LIN {X 0,Y 418.257,Z 234.886,A -85,B 0,C 180,E1 -9993.855,E2 -9993.855} C_VEL
LIN {X 0,Y 418.476,Z 234.858,A -85,B 0,C 180,E1 -9995.784,E2 -9995.784} C_VEL
LIN {X 0,Y 418.364,Z 234.87,A -85,B 0,C 180,E1 -9998.697,E2 -9998.697} C_VEL
LIN {X 0,Y 418.295,Z 234.879,A -85,B 0,C 180,E1 -10001.632,E2 -10001.632} C_VEL
LIN {X 0,Y 418.27,Z 234.881,A -85,B 0,C 180,E1 -10004.599,E2 -10004.599} C_VEL
LIN {X 0,Y 418.253,Z 234.884,A -85,B 0,C 180,E1 -10007.606,E2 -10007.606} C_VEL
LIN {X 0,Y 418.216,Z 234.886,A -85,B 0,C 180,E1 -10010.665,E2 -10010.665} C_VEL
LIN {X 0,Y 418.242,Z 234.885,A -85,B 0,C 180,E1 -10013.785,E2 -10013.785} C_VEL
LIN {X 0,Y 418.196,Z 234.889,A -85,B 0,C 180,E1 -10017.051,E2 -10017.051} C_VEL
LIN {X 0,Y 418.212,Z 234.887,A -85,B 0,C 180,E1 -10020.275,E2 -10020.275} C_VEL
LIN {X 0,Y 418.203,Z 234.887,A -85,B 0,C 180,E1 -10023.682,E2 -10023.682} C_VEL
LIN {X 0,Y 418.207,Z 234.887,A -85,B 0,C 180,E1 -10027.228,E2 -10027.228} C_VEL
LIN {X 0,Y 418.182,Z 234.887,A -85,B 0,C 180,E1 -10030.87,E2 -10030.87} C_VEL
LIN {X 0,Y 418.179,Z 234.883,A -85,B 0,C 180,E1 -10033.732,E2 -10033.732} C_VEL
LIN {X 0,Y 418.178,Z 234.894,A -85,B 0,C 180,E1 -10036.451,E2 -10036.451} C_VEL
LIN {X 0,Y 418.186,Z 234.885,A -85,B 0,C 180,E1 -10039.137,E2 -10039.137} C_VEL
LIN {X 0,Y 418.22,Z 234.877,A -85,B 0,C 180,E1 -10042.779,E2 -10042.779} C_VEL
LIN {X 0,Y 418.216,Z 234.886,A -85,B 0,C 180,E1 -10046.325,E2 -10046.325} C_VEL
LIN {X 0,Y 418.224,Z 234.873,A -85,B 0,C 180,E1 -10049.731,E2 -10049.731} C_VEL
LIN {X 0,Y 418.196,Z 234.877,A -85,B 0,C 180,E1 -10053.02,E2 -10053.02} C_VEL
LIN {X 0,Y 418.245,Z 234.882,A -85,B 0,C 180,E1 -10056.221,E2 -10056.221} C_VEL
LIN {X 0,Y 418.242,Z 234.884,A -85,B 0,C 180,E1 -10059.341,E2 -10059.341} C_VEL
LIN {X 0,Y 418.272,Z 234.856,A -85,B 0,C 180,E1 -10062.4,E2 -10062.4} C_VEL
LIN {X 0,Y 418.295,Z 234.87,A -85,B 0,C 180,E1 -10065.407,E2 -10065.407} C_VEL
LIN {X 0,Y 418.299,Z 234.876,A -85,B 0,C 180,E1 -10068.372,E2 -10068.372} C_VEL
LIN {X 0,Y 418.445,Z 234.844,A -85,B 0,C 180,E1 -10072.282,E2 -10072.282} C_VEL
LIN {X 0,Y 418.469,Z 234.837,A -85,B 0,C 180,E1 -10074.22,E2 -10074.22} C_VEL
LIN {X 0,Y 418.535,Z 234.848,A -85,B 0,C 180,E1 -10078.079,E2 -10078.079} C_VEL
LIN {X 0,Y 418.466,Z 234.853,A -85,B 0,C 180,E1 -10080.966,E2 -10080.966} C_VEL
LIN {X 0,Y 418.471,Z 234.845,A -85,B 0,C 180,E1 -10082.891,E2 -10082.891} C_VEL
LIN {X 0,Y 418.499,Z 234.832,A -85,B 0,C 180,E1 -10085.786,E2 -10085.786} C_VEL
LIN {X 0,Y 418.38,Z 234.87,A -85,B 0,C 180,E1 -10088.699,E2 -10088.699} C_VEL
LIN {X 0,Y 418.317,Z 234.873,A -85,B 0,C 180,E1 -10091.634,E2 -10091.634} C_VEL
LIN {X 0,Y 418.307,Z 234.865,A -85,B 0,C 180,E1 -10094.6,E2 -10094.6} C_VEL
LIN {X 0,Y 418.287,Z 234.874,A -85,B 0,C 180,E1 -10097.607,E2 -10097.607} C_VEL
LIN {X 0,Y 418.258,Z 234.887,A -85,B 0,C 180,E1 -10100.665,E2 -10100.665} C_VEL
LIN {X 0,Y 418.282,Z 234.863,A -85,B 0,C 180,E1 -10103.784,E2 -10103.784} C_VEL
LIN {X 0,Y 418.232,Z 234.889,A -85,B 0,C 180,E1 -10107.048,E2 -10107.048} C_VEL
LIN {X 0,Y 418.252,Z 234.877,A -85,B 0,C 180,E1 -10110.274,E2 -10110.274} C_VEL
LIN {X 0,Y 418.243,Z 234.886,A -85,B 0,C 180,E1 -10113.68,E2 -10113.68} C_VEL
LIN {X 0,Y 418.248,Z 234.881,A -85,B 0,C 180,E1 -10117.226,E2 -10117.226} C_VEL
LIN {X 0,Y 418.219,Z 234.887,A -85,B 0,C 180,E1 -10120.868,E2 -10120.868} C_VEL
LIN {X 0,Y 418.216,Z 234.891,A -85,B 0,C 180,E1 -10123.73,E2 -10123.73} C_VEL
LIN {X 0,Y 418.212,Z 234.885,A -85,B 0,C 180,E1 -10126.448,E2 -10126.448} C_VEL
LIN {X 0,Y 418.219,Z 234.887,A -85,B 0,C 180,E1 -10129.134,E2 -10129.134} C_VEL
LIN {X 0,Y 418.249,Z 234.884,A -85,B 0,C 180,E1 -10132.776,E2 -10132.776} C_VEL
LIN {X 0,Y 418.26,Z 234.88,A -85,B 0,C 180,E1 -10136.323,E2 -10136.323} C_VEL
LIN {X 0,Y 418.256,Z 234.882,A -85,B 0,C 180,E1 -10139.728,E2 -10139.728} C_VEL
LIN {X 0,Y 418.276,Z 234.882,A -85,B 0,C 180,E1 -10143.021,E2 -10143.021} C_VEL
LIN {X 0,Y 418.325,Z 235.179,A -85,B 0,C 180,E1 -10143.563,E2 -10143.563} C_VEL
LIN {X 0,Y 420.735,Z 247.292,A -85,B 0,C 180,E1 -10146.365,E2 -10146.365} C_VEL
LIN {X 0,Y 421.002,Z 250.418,A -85,B 0,C 180,E1 -10147.052,E2 -10147.052} C_VEL
LIN {X 0,Y 419.833,Z 267.822,A -85,B 0,C 180,E1 -10150.693,E2 -10150.693} C_VEL
LIN {X 0,Y 419.789,Z 269.662,A -85,B 0,C 180,E1 -10151.009,E2 -10151.009} C_VEL
LIN {X 0,Y 423.734,Z 293.591,A -85,B 0,C 180,E1 -10151.631,E2 -10151.631} C_VEL
LIN {X 0,Y 422.717,Z 377.028,A -85,B 0,C 180,E1 -10153.084,E2 -10153.084} C_VEL
LIN {X 0,Y 422.229,Z 390.307,A -85,B 0,C 180,E1 -10153.5,E2 -10153.5} C_VEL
LIN {X 0,Y 421.642,Z 403.053,A -85,B 0,C 180,E1 -10154.098,E2 -10154.098} C_VEL
LIN {X 0,Y 420.933,Z 415.178,A -85,B 0,C 180,E1 -10154.877,E2 -10154.877} C_VEL
LIN {X 0,Y 420.162,Z 427.115,A -85,B 0,C 180,E1 -10155.877,E2 -10155.877} C_VEL
LIN {X 0,Y 419.545,Z 437.113,A -85,B 0,C 180,E1 -10156.929,E2 -10156.929} C_VEL
LIN {X 0,Y 418.846,Z 446.446,A -85,B 0,C 180,E1 -10158.138,E2 -10158.138} C_VEL
LIN {X 0,Y 418.173,Z 455.483,A -85,B 0,C 180,E1 -10159.591,E2 -10159.591} C_VEL
LIN {X 0,Y 417.731,Z 462.762,A -85,B 0,C 180,E1 -10161.046,E2 -10161.046} C_VEL
LIN {X 0,Y 417.411,Z 467.677,A -85,B 0,C 180,E1 -10162.258,E2 -10162.258} C_VEL
LIN {X 0,Y 417.167,Z 472.465,A -85,B 0,C 180,E1 -10163.717,E2 -10163.717} C_VEL
LIN {X 0,Y 417.121,Z 476.104,A -85,B 0,C 180,E1 -10165.167,E2 -10165.167} C_VEL
LIN {X 0,Y 417.003,Z 477.99,A -85,B 0,C 180,E1 -10166.134,E2 -10166.134} C_VEL
LIN {X 0,Y 416.987,Z 479.414,A -85,B 0,C 180,E1 -10167.101,E2 -10167.101} C_VEL
LIN {X 0,Y 417.033,Z 480.426,A -85,B 0,C 180,E1 -10168.068,E2 -10168.068} C_VEL
LIN {X 0,Y 416.986,Z 481.283,A -85,B 0,C 180,E1 -10169.999,E2 -10169.999} C_VEL
LIN {X 0,Y 416.996,Z 481.089,A -85,B 0,C 180,E1 -10170.965,E2 -10170.965} C_VEL
LIN {X 0,Y 417.033,Z 480.493,A -85,B 0,C 180,E1 -10171.931,E2 -10171.931} C_VEL
LIN {X 0,Y 417.003,Z 478.128,A -85,B 0,C 180,E1 -10173.865,E2 -10173.865} C_VEL
LIN {X 0,Y 417.162,Z 475.214,A -85,B 0,C 180,E1 -10175.316,E2 -10175.316} C_VEL
LIN {X 0,Y 417.25,Z 471.268,A -85,B 0,C 180,E1 -10176.77,E2 -10176.77} C_VEL
LIN {X 0,Y 417.547,Z 466.19,A -85,B 0,C 180,E1 -10178.225,E2 -10178.225} C_VEL
LIN {X 0,Y 417.934,Z 459.8,A -85,B 0,C 180,E1 -10179.68,E2 -10179.68} C_VEL
LIN {X 0,Y 418.486,Z 451.815,A -85,B 0,C 180,E1 -10181.135,E2 -10181.135} C_VEL
LIN {X 0,Y 419.313,Z 441.896,A -85,B 0,C 180,E1 -10182.584,E2 -10182.584} C_VEL
LIN {X 0,Y 420.026,Z 431.811,A -85,B 0,C 180,E1 -10183.759,E2 -10183.759} C_VEL
LIN {X 0,Y 420.708,Z 421.199,A -85,B 0,C 180,E1 -10184.758,E2 -10184.758} C_VEL
LIN {X 0,Y 421.457,Z 409.943,A -85,B 0,C 180,E1 -10185.597,E2 -10185.597} C_VEL
LIN {X 0,Y 422.163,Z 397.246,A -85,B 0,C 180,E1 -10186.315,E2 -10186.315} C_VEL
LIN {X 0,Y 422.717,Z 383.65,A -85,B 0,C 180,E1 -10186.852,E2 -10186.852} C_VEL
LIN {X 0,Y 423.144,Z 369.847,A -85,B 0,C 180,E1 -10187.176,E2 -10187.176} C_VEL
LIN {X 0,Y 423.875,Z 292.546,A -85,B 0,C 180,E1 -10188.521,E2 -10188.521} C_VEL
LIN {X 0,Y 419.885,Z 269.167,A -85,B 0,C 180,E1 -10189.174,E2 -10189.174} C_VEL
LIN {X 0,Y 420.808,Z 253.629,A -85,B 0,C 180,E1 -10192.33,E2 -10192.33} C_VEL
LIN {X 0,Y 421,Z 248.821,A -85,B 0,C 180,E1 -10193.34,E2 -10193.34} C_VEL
LIN {X 0,Y 418.677,Z 236.536,A -85,B 0,C 180,E1 -10196.143,E2 -10196.143} C_VEL
LIN {X 0,Y 418.322,Z 234.908,A -85,B 0,C 180,E1 -10196.604,E2 -10196.604} C_VEL
LIN {X 0,Y 418.271,Z 234.885,A -85,B 0,C 180,E1 -10199.16,E2 -10199.16} C_VEL
LIN {X 0,Y 418.263,Z 234.884,A -85,B 0,C 180,E1 -10202.842,E2 -10202.842} C_VEL
LIN {X 0,Y 418.248,Z 234.882,A -85,B 0,C 180,E1 -10206.236,E2 -10206.236} C_VEL
LIN {X 0,Y 418.204,Z 234.887,A -85,B 0,C 180,E1 -10209.686,E2 -10209.686} C_VEL
LIN {X 0,Y 418.225,Z 234.891,A -85,B 0,C 180,E1 -10212.318,E2 -10212.318} C_VEL
LIN {X 0,Y 418.237,Z 234.884,A -85,B 0,C 180,E1 -10215.106,E2 -10215.106} C_VEL
LIN {X 0,Y 418.235,Z 234.886,A -85,B 0,C 180,E1 -10217.763,E2 -10217.763} C_VEL
LIN {X 0,Y 418.239,Z 234.88,A -85,B 0,C 180,E1 -10221.554,E2 -10221.554} C_VEL
LIN {X 0,Y 418.251,Z 234.882,A -85,B 0,C 180,E1 -10225.156,E2 -10225.156} C_VEL
LIN {X 0,Y 418.244,Z 234.882,A -85,B 0,C 180,E1 -10227.469,E2 -10227.469} C_VEL
LIN {X 0,Y 418.261,Z 234.885,A -85,B 0,C 180,E1 -10230.895,E2 -10230.895} C_VEL
LIN {X 0,Y 418.217,Z 234.885,A -85,B 0,C 180,E1 -10234.09,E2 -10234.09} C_VEL
LIN {X 0,Y 418.226,Z 234.885,A -85,B 0,C 180,E1 -10237.26,E2 -10237.26} C_VEL
LIN {X 0,Y 418.281,Z 234.879,A -85,B 0,C 180,E1 -10240.361,E2 -10240.361} C_VEL
LIN {X 0,Y 418.313,Z 234.879,A -85,B 0,C 180,E1 -10243.402,E2 -10243.402} C_VEL
LIN {X 0,Y 418.342,Z 234.868,A -85,B 0,C 180,E1 -10246.997,E2 -10246.997} C_VEL
LIN {X 0,Y 418.32,Z 234.872,A -85,B 0,C 180,E1 -10250.325,E2 -10250.325} C_VEL
LIN {X 0,Y 418.459,Z 234.859,A -85,B 0,C 180,E1 -10253.245,E2 -10253.245} C_VEL
LIN {X 0,Y 418.308,Z 234.88,A -85,B 0,C 180,E1 -10255.178,E2 -10255.178} C_VEL
LIN {X 0,Y 418.522,Z 234.85,A -85,B 0,C 180,E1 -10258.072,E2 -10258.072} C_VEL
LIN {X 0,Y 418.52,Z 234.851,A -85,B 0,C 180,E1 -10261.921,E2 -10261.921} C_VEL
LIN {X 0,Y 418.418,Z 234.859,A -85,B 0,C 180,E1 -10266.479,E2 -10266.479} C_VEL
LIN {X 0,Y 418.353,Z 234.868,A -85,B 0,C 180,E1 -10268.692,E2 -10268.692} C_VEL
LIN {X 0,Y 418.338,Z 234.871,A -85,B 0,C 180,E1 -10272.611,E2 -10272.611} C_VEL
LIN {X 0,Y 418.283,Z 234.882,A -85,B 0,C 180,E1 -10275.591,E2 -10275.591} C_VEL
LIN {X 0,Y 418.256,Z 234.885,A -85,B 0,C 180,E1 -10278.614,E2 -10278.614} C_VEL
LIN {X 0,Y 418.215,Z 234.89,A -85,B 0,C 180,E1 -10281.693,E2 -10281.693} C_VEL
LIN {X 0,Y 418.247,Z 234.883,A -85,B 0,C 180,E1 -10284.856,E2 -10284.856} C_VEL
LIN {X 0,Y 418.226,Z 234.886,A -85,B 0,C 180,E1 -10288.063,E2 -10288.063} C_VEL
LIN {X 0,Y 418.187,Z 234.89,A -85,B 0,C 180,E1 -10291.393,E2 -10291.393} C_VEL
LIN {X 0,Y 418.241,Z 234.886,A -85,B 0,C 180,E1 -10294.577,E2 -10294.577} C_VEL
LIN {X 0,Y 418.211,Z 234.888,A -85,B 0,C 180,E1 -10297.832,E2 -10297.832} C_VEL
LIN {X 0,Y 418.239,Z 234.888,A -85,B 0,C 180,E1 -10300.94,E2 -10300.94} C_VEL
LIN {X 0,Y 418.303,Z 235.044,A -85,B 0,C 180,E1 -10302.724,E2 -10302.724} C_VEL
LIN {X 0,Y 420.273,Z 244.859,A -85,B 0,C 180,E1 -10305.027,E2 -10305.027} C_VEL
LIN {X 0,Y 420.476,Z 249.038,A -85,B 0,C 180,E1 -10305.942,E2 -10305.942} C_VEL
LIN {X 0,Y 419.996,Z 258.446,A -85,B 0,C 180,E1 -10307.877,E2 -10307.877} C_VEL
LIN {X 0,Y 424.024,Z 279.663,A -85,B 0,C 180,E1 -10308.495,E2 -10308.495} C_VEL
LIN {X 0,Y 422.987,Z 365.547,A -85,B 0,C 180,E1 -10310.001,E2 -10310.001} C_VEL
LIN {X 0,Y 422.557,Z 379.31,A -85,B 0,C 180,E1 -10310.436,E2 -10310.436} C_VEL
LIN {X 0,Y 422.008,Z 392.261,A -85,B 0,C 180,E1 -10311.053,E2 -10311.053} C_VEL
LIN {X 0,Y 421.307,Z 404.921,A -85,B 0,C 180,E1 -10311.888,E2 -10311.888} C_VEL
LIN {X 0,Y 420.52,Z 416.351,A -85,B 0,C 180,E1 -10312.863,E2 -10312.863} C_VEL
LIN {X 0,Y 419.798,Z 425.954,A -85,B 0,C 180,E1 -10313.883,E2 -10313.883} C_VEL
LIN {X 0,Y 419.22,Z 434.271,A -85,B 0,C 180,E1 -10314.959,E2 -10314.959} C_VEL
LIN {X 0,Y 418.541,Z 443.069,A -85,B 0,C 180,E1 -10316.351,E2 -10316.351} C_VEL
LIN {X 0,Y 417.991,Z 450.165,A -85,B 0,C 180,E1 -10317.736,E2 -10317.736} C_VEL
LIN {X 0,Y 417.595,Z 456.913,A -85,B 0,C 180,E1 -10319.392,E2 -10319.392} C_VEL
LIN {X 0,Y 417.253,Z 462.266,A -85,B 0,C 180,E1 -10321.137,E2 -10321.137} C_VEL
LIN {X 0,Y 416.99,Z 466.192,A -85,B 0,C 180,E1 -10322.932,E2 -10322.932} C_VEL
LIN {X 0,Y 416.899,Z 467.831,A -85,B 0,C 180,E1 -10324.006,E2 -10324.006} C_VEL
LIN {X 0,Y 416.837,Z 469.291,A -85,B 0,C 180,E1 -10325.556,E2 -10325.556} C_VEL
LIN {X 0,Y 416.773,Z 469.714,A -85,B 0,C 180,E1 -10327.18,E2 -10327.18} C_VEL
LIN {X 0,Y 416.83,Z 469.386,A -85,B 0,C 180,E1 -10328.228,E2 -10328.228} C_VEL
LIN {X 0,Y 416.837,Z 468.631,A -85,B 0,C 180,E1 -10329.265,E2 -10329.265} C_VEL
LIN {X 0,Y 416.982,Z 466.785,A -85,B 0,C 180,E1 -10330.693,E2 -10330.693} C_VEL
LIN {X 0,Y 417.16,Z 463.519,A -85,B 0,C 180,E1 -10332.348,E2 -10332.348} C_VEL
LIN {X 0,Y 417.403,Z 458.75,A -85,B 0,C 180,E1 -10334.039,E2 -10334.039} C_VEL
LIN {X 0,Y 417.787,Z 452.809,A -85,B 0,C 180,E1 -10335.634,E2 -10335.634} C_VEL
LIN {X 0,Y 418.218,Z 446.156,A -85,B 0,C 180,E1 -10337.053,E2 -10337.053} C_VEL
LIN {X 0,Y 418.742,Z 438.489,A -85,B 0,C 180,E1 -10338.382,E2 -10338.382} C_VEL
LIN {X 0,Y 419.451,Z 428.69,A -85,B 0,C 180,E1 -10339.746,E2 -10339.746} C_VEL
LIN {X 0,Y 420.123,Z 419.264,A -85,B 0,C 180,E1 -10340.811,E2 -10340.811} C_VEL
LIN {X 0,Y 419.772,Z 414.556,A -85,B 0,C 180,E1 -10341.294,E2 -10341.294} C_VEL
LIN {X 0,Y 417.471,Z 406.719,A -85,B 0,C 180,E1 -10342.063,E2 -10342.063} C_VEL
LIN {X 0,Y 415.262,Z 398.464,A -85,B 0,C 180,E1 -10342.761,E2 -10342.761} C_VEL
LIN {X 0,Y 414.864,Z 393.162,A -85,B 0,C 180,E1 -10343.118,E2 -10343.118} C_VEL
LIN {X 0,Y 415.338,Z 382.041,A -85,B 0,C 180,E1 -10343.686,E2 -10343.686} C_VEL
LIN {X 0,Y 415.835,Z 368.781,A -85,B 0,C 180,E1 -10344.15,E2 -10344.15} C_VEL
LIN {X 0,Y 416.183,Z 350.094,A -85,B 0,C 180,E1 -10344.522,E2 -10344.522} C_VEL
LIN {X 0,Y 416.884,Z 280.038,A -85,B 0,C 180,E1 -10345.753,E2 -10345.753} C_VEL
LIN {X 0,Y 412.979,Z 258.958,A -85,B 0,C 180,E1 -10346.342,E2 -10346.342} C_VEL
LIN {X 0,Y 413.209,Z 254.351,A -85,B 0,C 180,E1 -10347.32,E2 -10347.32} C_VEL
LIN {X 0,Y 413.524,Z 247.973,A -85,B 0,C 180,E1 -10348.784,E2 -10348.784} C_VEL
LIN {X 0,Y 412.086,Z 239.005,A -85,B 0,C 180,E1 -10350.978,E2 -10350.978} C_VEL
LIN {X 0,Y 411.483,Z 235.781,A -85,B 0,C 180,E1 -10351.836,E2 -10351.836} C_VEL
LIN {X 0,Y 411.438,Z 235.734,A -85,B 0,C 180,E1 -10355.883,E2 -10355.883} C_VEL
LIN {X 0,Y 411.319,Z 235.748,A -85,B 0,C 180,E1 -10358.847,E2 -10358.847} C_VEL
LIN {X 0,Y 411.263,Z 235.752,A -85,B 0,C 180,E1 -10361.834,E2 -10361.834} C_VEL
LIN {X 0,Y 411.226,Z 235.758,A -85,B 0,C 180,E1 -10364.855,E2 -10364.855} C_VEL
LIN {X 0,Y 411.218,Z 235.765,A -85,B 0,C 180,E1 -10367.917,E2 -10367.917} C_VEL
LIN {X 0,Y 411.163,Z 235.764,A -85,B 0,C 180,E1 -10371.037,E2 -10371.037} C_VEL
LIN {X 0,Y 411.18,Z 235.763,A -85,B 0,C 180,E1 -10374.219,E2 -10374.219} C_VEL
LIN {X 0,Y 411.158,Z 235.767,A -85,B 0,C 180,E1 -10377.486,E2 -10377.486} C_VEL
LIN {X 0,Y 411.159,Z 235.766,A -85,B 0,C 180,E1 -10380.851,E2 -10380.851} C_VEL
LIN {X 0,Y 411.164,Z 235.762,A -85,B 0,C 180,E1 -10384.338,E2 -10384.338} C_VEL
LIN {X 0,Y 411.159,Z 235.768,A -85,B 0,C 180,E1 -10386.746,E2 -10386.746} C_VEL
LIN {X 0,Y 411.142,Z 235.768,A -85,B 0,C 180,E1 -10389.723,E2 -10389.723} C_VEL
LIN {X 0,Y 411.139,Z 235.762,A -85,B 0,C 180,E1 -10393.139,E2 -10393.139} C_VEL
LIN {X 0,Y 411.142,Z 235.767,A -85,B 0,C 180,E1 -10395.885,E2 -10395.885} C_VEL
LIN {X 0,Y 411.138,Z 235.76,A -85,B 0,C 180,E1 -10399.497,E2 -10399.497} C_VEL
LIN {X 0,Y 411.168,Z 235.75,A -85,B 0,C 180,E1 -10402.029,E2 -10402.029} C_VEL
LIN {X 0,Y 411.186,Z 235.767,A -85,B 0,C 180,E1 -10405.127,E2 -10405.127} C_VEL
LIN {X 0,Y 411.148,Z 235.763,A -85,B 0,C 180,E1 -10408.006,E2 -10408.006} C_VEL
LIN {X 0,Y 411.158,Z 235.75,A -85,B 0,C 180,E1 -10411.41,E2 -10411.41} C_VEL
LIN {X 0,Y 411.177,Z 235.761,A -85,B 0,C 180,E1 -10414.945,E2 -10414.945} C_VEL
LIN {X 0,Y 411.194,Z 235.761,A -85,B 0,C 180,E1 -10417.917,E2 -10417.917} C_VEL
LIN {X 0,Y 411.211,Z 235.749,A -85,B 0,C 180,E1 -10421.055,E2 -10421.055} C_VEL
LIN {X 0,Y 411.247,Z 235.746,A -85,B 0,C 180,E1 -10424.135,E2 -10424.135} C_VEL
LIN {X 0,Y 411.298,Z 235.747,A -85,B 0,C 180,E1 -10427.169,E2 -10427.169} C_VEL
LIN {X 0,Y 411.276,Z 235.749,A -85,B 0,C 180,E1 -10430.165,E2 -10430.165} C_VEL
LIN {X 0,Y 411.389,Z 235.719,A -85,B 0,C 180,E1 -10433.135,E2 -10433.135} C_VEL
LIN {X 0,Y 411.287,Z 235.731,A -85,B 0,C 180,E1 -10435.102,E2 -10435.102} C_VEL
LIN {X 0,Y 411.504,Z 235.723,A -85,B 0,C 180,E1 -10438.046,E2 -10438.046} C_VEL
LIN {X 0,Y 411.431,Z 235.729,A -85,B 0,C 180,E1 -10440.982,E2 -10440.982} C_VEL
LIN {X 0,Y 411.429,Z 235.722,A -85,B 0,C 180,E1 -10442.941,E2 -10442.941} C_VEL
LIN {X 0,Y 411.435,Z 235.726,A -85,B 0,C 180,E1 -10446.87,E2 -10446.87} C_VEL
LIN {X 0,Y 411.289,Z 235.749,A -85,B 0,C 180,E1 -10449.842,E2 -10449.842} C_VEL
LIN {X 0,Y 411.313,Z 235.74,A -85,B 0,C 180,E1 -10453.106,E2 -10453.106} C_VEL
LIN {X 0,Y 411.266,Z 235.747,A -85,B 0,C 180,E1 -10456.891,E2 -10456.891} C_VEL
LIN {X 0,Y 411.24,Z 235.756,A -85,B 0,C 180,E1 -10459.989,E2 -10459.989} C_VEL
LIN {X 0,Y 411.204,Z 235.75,A -85,B 0,C 180,E1 -10463.15,E2 -10463.15} C_VEL
LIN {X 0,Y 411.195,Z 235.758,A -85,B 0,C 180,E1 -10466.387,E2 -10466.387} C_VEL
LIN {X 0,Y 411.207,Z 235.756,A -85,B 0,C 180,E1 -10469.715,E2 -10469.715} C_VEL
LIN {X 0,Y 411.215,Z 235.759,A -85,B 0,C 180,E1 -10473.158,E2 -10473.158} C_VEL
LIN {X 0,Y 411.202,Z 235.757,A -85,B 0,C 180,E1 -10476.554,E2 -10476.554} C_VEL
LIN {X 0,Y 411.18,Z 235.768,A -85,B 0,C 180,E1 -10479.722,E2 -10479.722} C_VEL
LIN {X 0,Y 411.176,Z 235.759,A -85,B 0,C 180,E1 -10483.136,E2 -10483.136} C_VEL
LIN {X 0,Y 411.175,Z 235.765,A -85,B 0,C 180,E1 -10485.883,E2 -10485.883} C_VEL
LIN {X 0,Y 411.16,Z 235.765,A -85,B 0,C 180,E1 -10488.775,E2 -10488.775} C_VEL
LIN {X 0,Y 411.197,Z 235.765,A -85,B 0,C 180,E1 -10492.026,E2 -10492.026} C_VEL
LIN {X 0,Y 411.217,Z 235.763,A -85,B 0,C 180,E1 -10495.667,E2 -10495.667} C_VEL
LIN {X 0,Y 411.201,Z 235.761,A -85,B 0,C 180,E1 -10499.153,E2 -10499.153} C_VEL
LIN {X 0,Y 411.254,Z 235.761,A -85,B 0,C 180,E1 -10502.521,E2 -10502.521} C_VEL
LIN {X 0,Y 411.304,Z 235.978,A -85,B 0,C 180,E1 -10503.286,E2 -10503.286} C_VEL
LIN {X 0,Y 413.93,Z 249.498,A -85,B 0,C 180,E1 -10506.473,E2 -10506.473} C_VEL
LIN {X 0,Y 413.717,Z 255.587,A -85,B 0,C 180,E1 -10507.791,E2 -10507.791} C_VEL
LIN {X 0,Y 412.851,Z 269.407,A -85,B 0,C 180,E1 -10510.677,E2 -10510.677} C_VEL
LIN {X 0,Y 414.868,Z 281.394,A -85,B 0,C 180,E1 -10511.022,E2 -10511.022} C_VEL
LIN {X 0,Y 416.982,Z 294.541,A -85,B 0,C 180,E1 -10511.355,E2 -10511.355} C_VEL
LIN {X 0,Y 415.893,Z 377.561,A -85,B 0,C 180,E1 -10512.83,E2 -10512.83} C_VEL
LIN {X 0,Y 415.331,Z 391.388,A -85,B 0,C 180,E1 -10513.281,E2 -10513.281} C_VEL
LIN {X 0,Y 414.745,Z 403.809,A -85,B 0,C 180,E1 -10513.889,E2 -10513.889} C_VEL
LIN {X 0,Y 413.955,Z 416.487,A -85,B 0,C 180,E1 -10514.742,E2 -10514.742} C_VEL
LIN {X 0,Y 413.223,Z 427.367,A -85,B 0,C 180,E1 -10515.683,E2 -10515.683} C_VEL
LIN {X 0,Y 412.534,Z 437.926,A -85,B 0,C 180,E1 -10516.828,E2 -10516.828} C_VEL
LIN {X 0,Y 411.715,Z 447.892,A -85,B 0,C 180,E1 -10518.179,E2 -10518.179} C_VEL
LIN {X 0,Y 411.084,Z 456.668,A -85,B 0,C 180,E1 -10519.658,E2 -10519.658} C_VEL
LIN {X 0,Y 410.607,Z 463.663,A -85,B 0,C 180,E1 -10521.138,E2 -10521.138} C_VEL
LIN {X 0,Y 410.285,Z 469.262,A -85,B 0,C 180,E1 -10522.618,E2 -10522.618} C_VEL
LIN {X 0,Y 410.063,Z 473.658,A -85,B 0,C 180,E1 -10524.097,E2 -10524.097} C_VEL
LIN {X 0,Y 410.035,Z 475.98,A -85,B 0,C 180,E1 -10525.083,E2 -10525.083} C_VEL
LIN {X 0,Y 409.923,Z 477.872,A -85,B 0,C 180,E1 -10526.067,E2 -10526.067} C_VEL
LIN {X 0,Y 409.886,Z 479.303,A -85,B 0,C 180,E1 -10527.051,E2 -10527.051} C_VEL
LIN {X 0,Y 409.93,Z 480.319,A -85,B 0,C 180,E1 -10528.034,E2 -10528.034} C_VEL
LIN {X 0,Y 409.922,Z 480.945,A -85,B 0,C 180,E1 -10529.017,E2 -10529.017} C_VEL
LIN {X 0,Y 409.91,Z 481.183,A -85,B 0,C 180,E1 -10529.999,E2 -10529.999} C_VEL
LIN {X 0,Y 409.922,Z 480.996,A -85,B 0,C 180,E1 -10530.982,E2 -10530.982} C_VEL
LIN {X 0,Y 409.929,Z 480.403,A -85,B 0,C 180,E1 -10531.964,E2 -10531.964} C_VEL
LIN {X 0,Y 409.925,Z 478.046,A -85,B 0,C 180,E1 -10533.931,E2 -10533.931} C_VEL
LIN {X 0,Y 410.079,Z 475.138,A -85,B 0,C 180,E1 -10535.408,E2 -10535.408} C_VEL
LIN {X 0,Y 410.187,Z 471.199,A -85,B 0,C 180,E1 -10536.888,E2 -10536.888} C_VEL
LIN {X 0,Y 410.493,Z 466.128,A -85,B 0,C 180,E1 -10538.367,E2 -10538.367} C_VEL
LIN {X 0,Y 410.905,Z 459.751,A -85,B 0,C 180,E1 -10539.847,E2 -10539.847} C_VEL
LIN {X 0,Y 411.514,Z 451.775,A -85,B 0,C 180,E1 -10541.326,E2 -10541.326} C_VEL
LIN {X 0,Y 412.383,Z 441.868,A -85,B 0,C 180,E1 -10542.799,E2 -10542.799} C_VEL
LIN {X 0,Y 413.097,Z 431.339,A -85,B 0,C 180,E1 -10544.045,E2 -10544.045} C_VEL
LIN {X 0,Y 413.862,Z 421.211,A -85,B 0,C 180,E1 -10545.008,E2 -10545.008} C_VEL
LIN {X 0,Y 414.614,Z 409.981,A -85,B 0,C 180,E1 -10545.862,E2 -10545.862} C_VEL
LIN {X 0,Y 415.367,Z 397.349,A -85,B 0,C 180,E1 -10546.589,E2 -10546.589} C_VEL
LIN {X 0,Y 415.955,Z 383.839,A -85,B 0,C 180,E1 -10547.134,E2 -10547.134} C_VEL
LIN {X 0,Y 416.384,Z 370.314,A -85,B 0,C 180,E1 -10547.464,E2 -10547.464} C_VEL
LIN {X 0,Y 417.199,Z 293.585,A -85,B 0,C 180,E1 -10548.82,E2 -10548.82} C_VEL
LIN {X 0,Y 412.997,Z 269.348,A -85,B 0,C 180,E1 -10549.498,E2 -10549.498} C_VEL
LIN {X 0,Y 413.044,Z 267.047,A -85,B 0,C 180,E1 -10549.894,E2 -10549.894} C_VEL
LIN {X 0,Y 414.064,Z 252.374,A -85,B 0,C 180,E1 -10552.977,E2 -10552.977} C_VEL
LIN {X 0,Y 413.881,Z 248.977,A -85,B 0,C 180,E1 -10553.724,E2 -10553.724} C_VEL
LIN {X 0,Y 411.307,Z 235.976,A -85,B 0,C 180,E1 -10556.783,E2 -10556.783} C_VEL
LIN {X 0,Y 411.206,Z 235.763,A -85,B 0,C 180,E1 -10559.711,E2 -10559.711} C_VEL
LIN {X 0,Y 411.212,Z 235.763,A -85,B 0,C 180,E1 -10563.154,E2 -10563.154} C_VEL
LIN {X 0,Y 411.196,Z 235.759,A -85,B 0,C 180,E1 -10566.55,E2 -10566.55} C_VEL
LIN {X 0,Y 411.173,Z 235.763,A -85,B 0,C 180,E1 -10569.718,E2 -10569.718} C_VEL
LIN {X 0,Y 411.173,Z 235.763,A -85,B 0,C 180,E1 -10573.132,E2 -10573.132} C_VEL
LIN {X 0,Y 411.17,Z 235.766,A -85,B 0,C 180,E1 -10575.879,E2 -10575.879} C_VEL
LIN {X 0,Y 411.155,Z 235.77,A -85,B 0,C 180,E1 -10578.771,E2 -10578.771} C_VEL
LIN {X 0,Y 411.187,Z 235.761,A -85,B 0,C 180,E1 -10582.023,E2 -10582.023} C_VEL
LIN {X 0,Y 411.204,Z 235.76,A -85,B 0,C 180,E1 -10585.121,E2 -10585.121} C_VEL
LIN {X 0,Y 411.165,Z 235.765,A -85,B 0,C 180,E1 -10588,E2 -10588} C_VEL
LIN {X 0,Y 411.175,Z 235.763,A -85,B 0,C 180,E1 -10591.404,E2 -10591.404} C_VEL
LIN {X 0,Y 411.187,Z 235.768,A -85,B 0,C 180,E1 -10594.938,E2 -10594.938} C_VEL
LIN {X 0,Y 411.201,Z 235.757,A -85,B 0,C 180,E1 -10597.91,E2 -10597.91} C_VEL
LIN {X 0,Y 411.216,Z 235.758,A -85,B 0,C 180,E1 -10601.048,E2 -10601.048} C_VEL
LIN {X 0,Y 411.248,Z 235.755,A -85,B 0,C 180,E1 -10604.129,E2 -10604.129} C_VEL
LIN {X 0,Y 411.299,Z 235.747,A -85,B 0,C 180,E1 -10607.163,E2 -10607.163} C_VEL
LIN {X 0,Y 411.275,Z 235.749,A -85,B 0,C 180,E1 -10610.158,E2 -10610.158} C_VEL
LIN {X 0,Y 411.425,Z 235.734,A -85,B 0,C 180,E1 -10613.129,E2 -10613.129} C_VEL
LIN {X 0,Y 411.281,Z 235.754,A -85,B 0,C 180,E1 -10615.095,E2 -10615.095} C_VEL
LIN {X 0,Y 411.491,Z 235.726,A -85,B 0,C 180,E1 -10618.039,E2 -10618.039} C_VEL
LIN {X 0,Y 411.489,Z 235.727,A -85,B 0,C 180,E1 -10621.954,E2 -10621.954} C_VEL
LIN {X 0,Y 411.368,Z 235.737,A -85,B 0,C 180,E1 -10626.477,E2 -10626.477} C_VEL
LIN {X 0,Y 411.293,Z 235.748,A -85,B 0,C 180,E1 -10628.843,E2 -10628.843} C_VEL
LIN {X 0,Y 411.259,Z 235.76,A -85,B 0,C 180,E1 -10631.83,E2 -10631.83} C_VEL
LIN {X 0,Y 411.241,Z 235.757,A -85,B 0,C 180,E1 -10634.849,E2 -10634.849} C_VEL
LIN {X 0,Y 411.227,Z 235.76,A -85,B 0,C 180,E1 -10637.912,E2 -10637.912} C_VEL
LIN {X 0,Y 411.177,Z 235.764,A -85,B 0,C 180,E1 -10641.031,E2 -10641.031} C_VEL
LIN {X 0,Y 411.192,Z 235.768,A -85,B 0,C 180,E1 -10644.213,E2 -10644.213} C_VEL
LIN {X 0,Y 411.167,Z 235.766,A -85,B 0,C 180,E1 -10647.48,E2 -10647.48} C_VEL
LIN {X 0,Y 411.165,Z 235.768,A -85,B 0,C 180,E1 -10650.845,E2 -10650.845} C_VEL
LIN {X 0,Y 411.181,Z 235.767,A -85,B 0,C 180,E1 -10654.33,E2 -10654.33} C_VEL
LIN {X 0,Y 411.178,Z 235.765,A -85,B 0,C 180,E1 -10657.97,E2 -10657.97} C_VEL
LIN {X 0,Y 411.183,Z 235.768,A -85,B 0,C 180,E1 -10661.233,E2 -10661.233} C_VEL
LIN {X 0,Y 411.256,Z 235.96,A -85,B 0,C 180,E1 -10662.452,E2 -10662.452} C_VEL
LIN {X 0,Y 413.507,Z 247.488,A -85,B 0,C 180,E1 -10665.194,E2 -10665.194} C_VEL
LIN {X 0,Y 413.299,Z 254.821,A -85,B 0,C 180,E1 -10666.781,E2 -10666.781} C_VEL
LIN {X 0,Y 413.17,Z 258.636,A -85,B 0,C 180,E1 -10667.537,E2 -10667.537} C_VEL
LIN {X 0,Y 417.351,Z 280.584,A -85,B 0,C 180,E1 -10668.19,E2 -10668.19} C_VEL
LIN {X 0,Y 416.189,Z 366.364,A -85,B 0,C 180,E1 -10669.723,E2 -10669.723} C_VEL
LIN {X 0,Y 415.757,Z 380.018,A -85,B 0,C 180,E1 -10670.172,E2 -10670.172} C_VEL
LIN {X 0,Y 415.23,Z 392.101,A -85,B 0,C 180,E1 -10670.76,E2 -10670.76} C_VEL
LIN {X 0,Y 414.629,Z 403.053,A -85,B 0,C 180,E1 -10671.472,E2 -10671.472} C_VEL
LIN {X 0,Y 413.787,Z 414.416,A -85,B 0,C 180,E1 -10672.419,E2 -10672.419} C_VEL
LIN {X 0,Y 412.93,Z 425.552,A -85,B 0,C 180,E1 -10673.591,E2 -10673.591} C_VEL
LIN {X 0,Y 412.184,Z 435.562,A -85,B 0,C 180,E1 -10674.919,E2 -10674.919} C_VEL
LIN {X 0,Y 411.487,Z 443.872,A -85,B 0,C 180,E1 -10676.285,E2 -10676.285} C_VEL
LIN {X 0,Y 410.931,Z 450.847,A -85,B 0,C 180,E1 -10677.694,E2 -10677.694} C_VEL
LIN {X 0,Y 410.565,Z 456.474,A -85,B 0,C 180,E1 -10679.102,E2 -10679.102} C_VEL
LIN {X 0,Y 410.206,Z 462.03,A -85,B 0,C 180,E1 -10680.89,E2 -10680.89} C_VEL
LIN {X 0,Y 410.012,Z 465.535,A -85,B 0,C 180,E1 -10682.433,E2 -10682.433} C_VEL
LIN {X 0,Y 409.837,Z 467.351,A -85,B 0,C 180,E1 -10683.523,E2 -10683.523} C_VEL
LIN {X 0,Y 409.734,Z 469.303,A -85,B 0,C 180,E1 -10685.367,E2 -10685.367} C_VEL
LIN {X 0,Y 409.693,Z 469.807,A -85,B 0,C 180,E1 -10686.763,E2 -10686.763} C_VEL
LIN {X 0,Y 409.692,Z 469.672,A -85,B 0,C 180,E1 -10687.857,E2 -10687.857} C_VEL
LIN {X 0,Y 409.73,Z 469.06,A -85,B 0,C 180,E1 -10688.888,E2 -10688.888} C_VEL
LIN {X 0,Y 409.869,Z 467.155,A -85,B 0,C 180,E1 -10690.56,E2 -10690.56} C_VEL
LIN {X 0,Y 410.019,Z 464.481,A -85,B 0,C 180,E1 -10692.03,E2 -10692.03} C_VEL
LIN {X 0,Y 410.218,Z 460.513,A -85,B 0,C 180,E1 -10693.601,E2 -10693.601} C_VEL
LIN {X 0,Y 410.555,Z 455.461,A -85,B 0,C 180,E1 -10695.122,E2 -10695.122} C_VEL
LIN {X 0,Y 410.997,Z 449.104,A -85,B 0,C 180,E1 -10696.635,E2 -10696.635} C_VEL
LIN {X 0,Y 411.584,Z 440.919,A -85,B 0,C 180,E1 -10698.177,E2 -10698.177} C_VEL
LIN {X 0,Y 412.207,Z 432.636,A -85,B 0,C 180,E1 -10699.44,E2 -10699.44} C_VEL
LIN {X 0,Y 413.001,Z 422.379,A -85,B 0,C 180,E1 -10700.712,E2 -10700.712} C_VEL
LIN {X 0,Y 413.796,Z 411.053,A -85,B 0,C 180,E1 -10701.823,E2 -10701.823} C_VEL
LIN {X 0,Y 414.549,Z 399.759,A -85,B 0,C 180,E1 -10702.696,E2 -10702.696} C_VEL
LIN {X 0,Y 414.864,Z 393.162,A -85,B 0,C 180,E1 -10703.118,E2 -10703.118} C_VEL
LIN {X 0,Y 414.381,Z 389.563,A -85,B 0,C 180,E1 -10703.354,E2 -10703.354} C_VEL
LIN {X 0,Y 409.267,Z 378.214,A -85,B 0,C 180,E1 -10704.099,E2 -10704.099} C_VEL
LIN {X 0,Y 408.871,Z 374.429,A -85,B 0,C 180,E1 -10704.255,E2 -10704.255} C_VEL
LIN {X 0,Y 409.232,Z 361.718,A -85,B 0,C 180,E1 -10704.599,E2 -10704.599} C_VEL
LIN {X 0,Y 410.187,Z 281.4,A -85,B 0,C 180,E1 -10706.032,E2 -10706.032} C_VEL
LIN {X 0,Y 406.081,Z 259.104,A -85,B 0,C 180,E1 -10706.662,E2 -10706.662} C_VEL
LIN {X 0,Y 406.283,Z 255.054,A -85,B 0,C 180,E1 -10707.522,E2 -10707.522} C_VEL
LIN {X 0,Y 406.518,Z 248.699,A -85,B 0,C 180,E1 -10709.01,E2 -10709.01} C_VEL
LIN {X 0,Y 405.213,Z 240.733,A -85,B 0,C 180,E1 -10710.995,E2 -10710.995} C_VEL
LIN {X 0,Y 404.449,Z 236.659,A -85,B 0,C 180,E1 -10712.086,E2 -10712.086} C_VEL
LIN {X 0,Y 404.386,Z 236.612,A -85,B 0,C 180,E1 -10715.986,E2 -10715.986} C_VEL
LIN {X 0,Y 404.256,Z 236.627,A -85,B 0,C 180,E1 -10719.003,E2 -10719.003} C_VEL
LIN {X 0,Y 404.234,Z 236.625,A -85,B 0,C 180,E1 -10722.043,E2 -10722.043} C_VEL
LIN {X 0,Y 404.172,Z 236.638,A -85,B 0,C 180,E1 -10725.12,E2 -10725.12} C_VEL
LIN {X 0,Y 404.176,Z 236.638,A -85,B 0,C 180,E1 -10728.24,E2 -10728.24} C_VEL
LIN {X 0,Y 404.105,Z 236.645,A -85,B 0,C 180,E1 -10731.422,E2 -10731.422} C_VEL
LIN {X 0,Y 404.132,Z 236.64,A -85,B 0,C 180,E1 -10734.669,E2 -10734.669} C_VEL
LIN {X 0,Y 404.1,Z 236.647,A -85,B 0,C 180,E1 -10738.008,E2 -10738.008} C_VEL
LIN {X 0,Y 404.115,Z 236.642,A -85,B 0,C 180,E1 -10740.288,E2 -10740.288} C_VEL
LIN {X 0,Y 404.11,Z 236.644,A -85,B 0,C 180,E1 -10743.816,E2 -10743.816} C_VEL
LIN {X 0,Y 404.105,Z 236.646,A -85,B 0,C 180,E1 -10746.877,E2 -10746.877} C_VEL
LIN {X 0,Y 404.092,Z 236.648,A -85,B 0,C 180,E1 -10750.078,E2 -10750.078} C_VEL
LIN {X 0,Y 404.118,Z 236.636,A -85,B 0,C 180,E1 -10753.086,E2 -10753.086} C_VEL
LIN {X 0,Y 404.098,Z 236.644,A -85,B 0,C 180,E1 -10755.926,E2 -10755.926} C_VEL
LIN {X 0,Y 404.082,Z 236.65,A -85,B 0,C 180,E1 -10758.636,E2 -10758.636} C_VEL
LIN {X 0,Y 404.122,Z 236.629,A -85,B 0,C 180,E1 -10761.499,E2 -10761.499} C_VEL
LIN {X 0,Y 404.158,Z 236.64,A -85,B 0,C 180,E1 -10764.987,E2 -10764.987} C_VEL
LIN {X 0,Y 404.122,Z 236.638,A -85,B 0,C 180,E1 -10768.447,E2 -10768.447} C_VEL
LIN {X 0,Y 404.135,Z 236.625,A -85,B 0,C 180,E1 -10770.866,E2 -10770.866} C_VEL
LIN {X 0,Y 404.143,Z 236.635,A -85,B 0,C 180,E1 -10774.727,E2 -10774.727} C_VEL
LIN {X 0,Y 404.157,Z 236.642,A -85,B 0,C 180,E1 -10777.512,E2 -10777.512} C_VEL
LIN {X 0,Y 404.155,Z 236.626,A -85,B 0,C 180,E1 -10780.711,E2 -10780.711} C_VEL
LIN {X 0,Y 404.215,Z 236.616,A -85,B 0,C 180,E1 -10783.852,E2 -10783.852} C_VEL
LIN {X 0,Y 404.28,Z 236.62,A -85,B 0,C 180,E1 -10786.943,E2 -10786.943} C_VEL
LIN {X 0,Y 404.243,Z 236.627,A -85,B 0,C 180,E1 -10789.992,E2 -10789.992} C_VEL
LIN {X 0,Y 404.34,Z 236.597,A -85,B 0,C 180,E1 -10793.015,E2 -10793.015} C_VEL
LIN {X 0,Y 404.258,Z 236.606,A -85,B 0,C 180,E1 -10795.017,E2 -10795.017} C_VEL
LIN {X 0,Y 404.473,Z 236.598,A -85,B 0,C 180,E1 -10798.012,E2 -10798.012} C_VEL
LIN {X 0,Y 404.397,Z 236.605,A -85,B 0,C 180,E1 -10800.999,E2 -10800.999} C_VEL
LIN {X 0,Y 404.363,Z 236.602,A -85,B 0,C 180,E1 -10802.992,E2 -10802.992} C_VEL
LIN {X 0,Y 404.396,Z 236.589,A -85,B 0,C 180,E1 -10805.989,E2 -10805.989} C_VEL
LIN {X 0,Y 404.267,Z 236.625,A -85,B 0,C 180,E1 -10809.005,E2 -10809.005} C_VEL
LIN {X 0,Y 404.261,Z 236.625,A -85,B 0,C 180,E1 -10812.044,E2 -10812.044} C_VEL
LIN {X 0,Y 404.211,Z 236.616,A -85,B 0,C 180,E1 -10815.121,E2 -10815.121} C_VEL
LIN {X 0,Y 404.213,Z 236.628,A -85,B 0,C 180,E1 -10818.241,E2 -10818.241} C_VEL
LIN {X 0,Y 404.147,Z 236.637,A -85,B 0,C 180,E1 -10821.422,E2 -10821.422} C_VEL
LIN {X 0,Y 404.17,Z 236.624,A -85,B 0,C 180,E1 -10824.669,E2 -10824.669} C_VEL
LIN {X 0,Y 404.13,Z 236.641,A -85,B 0,C 180,E1 -10828.007,E2 -10828.007} C_VEL
LIN {X 0,Y 404.154,Z 236.633,A -85,B 0,C 180,E1 -10830.287,E2 -10830.287} C_VEL
LIN {X 0,Y 404.149,Z 236.641,A -85,B 0,C 180,E1 -10833.815,E2 -10833.815} C_VEL
LIN {X 0,Y 404.145,Z 236.638,A -85,B 0,C 180,E1 -10836.876,E2 -10836.876} C_VEL
LIN {X 0,Y 404.128,Z 236.643,A -85,B 0,C 180,E1 -10840.076,E2 -10840.076} C_VEL
LIN {X 0,Y 404.156,Z 236.633,A -85,B 0,C 180,E1 -10843.083,E2 -10843.083} C_VEL
LIN {X 0,Y 404.132,Z 236.642,A -85,B 0,C 180,E1 -10845.923,E2 -10845.923} C_VEL
LIN {X 0,Y 404.115,Z 236.643,A -85,B 0,C 180,E1 -10848.634,E2 -10848.634} C_VEL
LIN {X 0,Y 404.151,Z 236.643,A -85,B 0,C 180,E1 -10851.496,E2 -10851.496} C_VEL
LIN {X 0,Y 404.196,Z 236.635,A -85,B 0,C 180,E1 -10854.984,E2 -10854.984} C_VEL
LIN {X 0,Y 404.151,Z 236.642,A -85,B 0,C 180,E1 -10858.443,E2 -10858.443} C_VEL
LIN {X 0,Y 404.199,Z 236.635,A -85,B 0,C 180,E1 -10862,E2 -10862} C_VEL
LIN {X 0,Y 404.251,Z 236.853,A -85,B 0,C 180,E1 -10863.023,E2 -10863.023} C_VEL
LIN {X 0,Y 406.647,Z 248.969,A -85,B 0,C 180,E1 -10865.948,E2 -10865.948} C_VEL
LIN {X 0,Y 407.081,Z 252.998,A -85,B 0,C 180,E1 -10866.873,E2 -10866.873} C_VEL
LIN {X 0,Y 405.938,Z 269.125,A -85,B 0,C 180,E1 -10870.335,E2 -10870.335} C_VEL
LIN {X 0,Y 406.589,Z 273.393,A -85,B 0,C 180,E1 -10870.496,E2 -10870.496} C_VEL
LIN {X 0,Y 410.2,Z 295.407,A -85,B 0,C 180,E1 -10871.068,E2 -10871.068} C_VEL
LIN {X 0,Y 409.118,Z 376.957,A -85,B 0,C 180,E1 -10872.537,E2 -10872.537} C_VEL
LIN {X 0,Y 408.598,Z 390.189,A -85,B 0,C 180,E1 -10872.965,E2 -10872.965} C_VEL
LIN {X 0,Y 407.917,Z 403.47,A -85,B 0,C 180,E1 -10873.612,E2 -10873.612} C_VEL
LIN {X 0,Y 407.18,Z 414.624,A -85,B 0,C 180,E1 -10874.353,E2 -10874.353} C_VEL
LIN {X 0,Y 406.364,Z 426.617,A -85,B 0,C 180,E1 -10875.386,E2 -10875.386} C_VEL
LIN {X 0,Y 405.631,Z 436.675,A -85,B 0,C 180,E1 -10876.472,E2 -10876.472} C_VEL
LIN {X 0,Y 404.898,Z 446.069,A -85,B 0,C 180,E1 -10877.723,E2 -10877.723} C_VEL
LIN {X 0,Y 404.146,Z 455.138,A -85,B 0,C 180,E1 -10879.225,E2 -10879.225} C_VEL
LIN {X 0,Y 403.626,Z 462.444,A -85,B 0,C 180,E1 -10880.731,E2 -10880.731} C_VEL
LIN {X 0,Y 403.307,Z 467.386,A -85,B 0,C 180,E1 -10881.986,E2 -10881.986} C_VEL
LIN {X 0,Y 402.988,Z 472.961,A -85,B 0,C 180,E1 -10883.767,E2 -10883.767} C_VEL
LIN {X 0,Y 402.95,Z 475.855,A -85,B 0,C 180,E1 -10884.996,E2 -10884.996} C_VEL
LIN {X 0,Y 402.846,Z 477.751,A -85,B 0,C 180,E1 -10885.998,E2 -10885.998} C_VEL
LIN {X 0,Y 402.788,Z 479.191,A -85,B 0,C 180,E1 -10886.999,E2 -10886.999} C_VEL
LIN {X 0,Y 402.826,Z 480.211,A -85,B 0,C 180,E1 -10888,E2 -10888} C_VEL
LIN {X 0,Y 402.849,Z 480.841,A -85,B 0,C 180,E1 -10889,E2 -10889} C_VEL
LIN {X 0,Y 402.836,Z 481.084,A -85,B 0,C 180,E1 -10889.999,E2 -10889.999} C_VEL
LIN {X 0,Y 402.849,Z 480.903,A -85,B 0,C 180,E1 -10890.999,E2 -10890.999} C_VEL
LIN {X 0,Y 402.826,Z 480.313,A -85,B 0,C 180,E1 -10891.999,E2 -10891.999} C_VEL
LIN {X 0,Y 402.849,Z 477.963,A -85,B 0,C 180,E1 -10894.001,E2 -10894.001} C_VEL
LIN {X 0,Y 402.976,Z 475.062,A -85,B 0,C 180,E1 -10895.503,E2 -10895.503} C_VEL
LIN {X 0,Y 403.11,Z 471.129,A -85,B 0,C 180,E1 -10897.009,E2 -10897.009} C_VEL
LIN {X 0,Y 403.453,Z 466.066,A -85,B 0,C 180,E1 -10898.514,E2 -10898.514} C_VEL
LIN {X 0,Y 403.888,Z 459.7,A -85,B 0,C 180,E1 -10900.02,E2 -10900.02} C_VEL
LIN {X 0,Y 404.536,Z 451.735,A -85,B 0,C 180,E1 -10901.524,E2 -10901.524} C_VEL
LIN {X 0,Y 405.44,Z 441.84,A -85,B 0,C 180,E1 -10903.022,E2 -10903.022} C_VEL
LIN {X 0,Y 406.137,Z 432.299,A -85,B 0,C 180,E1 -10904.186,E2 -10904.186} C_VEL
LIN {X 0,Y 406.877,Z 422.665,A -85,B 0,C 180,E1 -10905.144,E2 -10905.144} C_VEL
LIN {X 0,Y 407.702,Z 411.816,A -85,B 0,C 180,E1 -10906.009,E2 -10906.009} C_VEL
LIN {X 0,Y 408.409,Z 399.861,A -85,B 0,C 180,E1 -10906.751,E2 -10906.751} C_VEL
LIN {X 0,Y 409.098,Z 386.854,A -85,B 0,C 180,E1 -10907.334,E2 -10907.334} C_VEL
LIN {X 0,Y 409.529,Z 373.962,A -85,B 0,C 180,E1 -10907.701,E2 -10907.701} C_VEL
LIN {X 0,Y 410.541,Z 294.671,A -85,B 0,C 180,E1 -10909.131,E2 -10909.131} C_VEL
LIN {X 0,Y 406.32,Z 270.523,A -85,B 0,C 180,E1 -10909.807,E2 -10909.807} C_VEL
LIN {X 0,Y 406.063,Z 268.841,A -85,B 0,C 180,E1 -10909.897,E2 -10909.897} C_VEL
LIN {X 0,Y 407.163,Z 253.578,A -85,B 0,C 180,E1 -10913.121,E2 -10913.121} C_VEL
LIN {X 0,Y 406.772,Z 249.447,A -85,B 0,C 180,E1 -10914.056,E2 -10914.056} C_VEL
LIN {X 0,Y 404.436,Z 237.713,A -85,B 0,C 180,E1 -10916.859,E2 -10916.859} C_VEL
LIN {X 0,Y 404.251,Z 236.662,A -85,B 0,C 180,E1 -10917.186,E2 -10917.186} C_VEL
LIN {X 0,Y 404.151,Z 236.644,A -85,B 0,C 180,E1 -10920.283,E2 -10920.283} C_VEL
LIN {X 0,Y 404.15,Z 236.64,A -85,B 0,C 180,E1 -10923.81,E2 -10923.81} C_VEL
LIN {X 0,Y 404.139,Z 236.638,A -85,B 0,C 180,E1 -10926.872,E2 -10926.872} C_VEL
LIN {X 0,Y 404.121,Z 236.639,A -85,B 0,C 180,E1 -10930.073,E2 -10930.073} C_VEL
LIN {X 0,Y 404.153,Z 236.637,A -85,B 0,C 180,E1 -10933.081,E2 -10933.081} C_VEL
LIN {X 0,Y 404.15,Z 236.641,A -85,B 0,C 180,E1 -10935.923,E2 -10935.923} C_VEL
LIN {X 0,Y 404.11,Z 236.646,A -85,B 0,C 180,E1 -10938.631,E2 -10938.631} C_VEL
LIN {X 0,Y 404.142,Z 236.636,A -85,B 0,C 180,E1 -10941.492,E2 -10941.492} C_VEL
LIN {X 0,Y 404.175,Z 236.636,A -85,B 0,C 180,E1 -10944.98,E2 -10944.98} C_VEL
LIN {X 0,Y 404.139,Z 236.641,A -85,B 0,C 180,E1 -10948.44,E2 -10948.44} C_VEL
LIN {X 0,Y 404.151,Z 236.643,A -85,B 0,C 180,E1 -10950.86,E2 -10950.86} C_VEL
LIN {X 0,Y 404.152,Z 236.643,A -85,B 0,C 180,E1 -10954.72,E2 -10954.72} C_VEL
LIN {X 0,Y 404.165,Z 236.635,A -85,B 0,C 180,E1 -10957.505,E2 -10957.505} C_VEL
LIN {X 0,Y 404.159,Z 236.641,A -85,B 0,C 180,E1 -10960.704,E2 -10960.704} C_VEL
LIN {X 0,Y 404.216,Z 236.631,A -85,B 0,C 180,E1 -10963.845,E2 -10963.845} C_VEL
LIN {X 0,Y 404.279,Z 236.619,A -85,B 0,C 180,E1 -10966.936,E2 -10966.936} C_VEL
LIN {X 0,Y 404.242,Z 236.626,A -85,B 0,C 180,E1 -10969.985,E2 -10969.985} C_VEL
LIN {X 0,Y 404.375,Z 236.61,A -85,B 0,C 180,E1 -10973.009,E2 -10973.009} C_VEL
LIN {X 0,Y 404.254,Z 236.629,A -85,B 0,C 180,E1 -10975.01,E2 -10975.01} C_VEL
LIN {X 0,Y 404.46,Z 236.602,A -85,B 0,C 180,E1 -10978.005,E2 -10978.005} C_VEL
LIN {X 0,Y 404.458,Z 236.603,A -85,B 0,C 180,E1 -10981.988,E2 -10981.988} C_VEL
LIN {X 0,Y 404.321,Z 236.615,A -85,B 0,C 180,E1 -10986.474,E2 -10986.474} C_VEL
LIN {X 0,Y 404.242,Z 236.626,A -85,B 0,C 180,E1 -10988.998,E2 -10988.998} C_VEL
LIN {X 0,Y 404.234,Z 236.633,A -85,B 0,C 180,E1 -10992.038,E2 -10992.038} C_VEL
LIN {X 0,Y 404.188,Z 236.636,A -85,B 0,C 180,E1 -10995.115,E2 -10995.115} C_VEL
LIN {X 0,Y 404.186,Z 236.641,A -85,B 0,C 180,E1 -10998.235,E2 -10998.235} C_VEL
LIN {X 0,Y 404.119,Z 236.644,A -85,B 0,C 180,E1 -11001.416,E2 -11001.416} C_VEL
LIN {X 0,Y 404.144,Z 236.641,A -85,B 0,C 180,E1 -11004.663,E2 -11004.663} C_VEL
LIN {X 0,Y 404.108,Z 236.644,A -85,B 0,C 180,E1 -11008.001,E2 -11008.001} C_VEL
LIN {X 0,Y 404.121,Z 236.647,A -85,B 0,C 180,E1 -11010.282,E2 -11010.282} C_VEL
LIN {X 0,Y 404.121,Z 236.646,A -85,B 0,C 180,E1 -11013.809,E2 -11013.809} C_VEL
LIN {X 0,Y 404.114,Z 236.646,A -85,B 0,C 180,E1 -11016.873,E2 -11016.873} C_VEL
LIN {X 0,Y 404.14,Z 236.645,A -85,B 0,C 180,E1 -11020.081,E2 -11020.081} C_VEL
LIN {X 0,Y 404.206,Z 236.72,A -85,B 0,C 180,E1 -11022.099,E2 -11022.099} C_VEL
LIN {X 0,Y 405.278,Z 242.084,A -85,B 0,C 180,E1 -11023.462,E2 -11023.462} C_VEL
LIN {X 0,Y 406.688,Z 250.081,A -85,B 0,C 180,E1 -11025.346,E2 -11025.346} C_VEL
LIN {X 0,Y 406.272,Z 258.551,A -85,B 0,C 180,E1 -11027.151,E2 -11027.151} C_VEL
LIN {X 0,Y 407.057,Z 262.671,A -85,B 0,C 180,E1 -11027.327,E2 -11027.327} C_VEL
LIN {X 0,Y 410.711,Z 282.156,A -85,B 0,C 180,E1 -11027.885,E2 -11027.885} C_VEL
LIN {X 0,Y 409.457,Z 366.408,A -85,B 0,C 180,E1 -11029.412,E2 -11029.412} C_VEL
LIN {X 0,Y 409,Z 379.932,A -85,B 0,C 180,E1 -11029.862,E2 -11029.862} C_VEL
LIN {X 0,Y 408.466,Z 392.062,A -85,B 0,C 180,E1 -11030.462,E2 -11030.462} C_VEL
LIN {X 0,Y 407.795,Z 403.521,A -85,B 0,C 180,E1 -11031.221,E2 -11031.221} C_VEL
LIN {X 0,Y 406.901,Z 414.826,A -85,B 0,C 180,E1 -11032.184,E2 -11032.184} C_VEL
LIN {X 0,Y 406.041,Z 425.557,A -85,B 0,C 180,E1 -11033.336,E2 -11033.336} C_VEL
LIN {X 0,Y 405.307,Z 434.872,A -85,B 0,C 180,E1 -11034.577,E2 -11034.577} C_VEL
LIN {X 0,Y 404.589,Z 443.134,A -85,B 0,C 180,E1 -11035.931,E2 -11035.931} C_VEL
LIN {X 0,Y 403.965,Z 450.255,A -85,B 0,C 180,E1 -11037.364,E2 -11037.364} C_VEL
LIN {X 0,Y 403.495,Z 457.115,A -85,B 0,C 180,E1 -11039.102,E2 -11039.102} C_VEL
LIN {X 0,Y 403.138,Z 462.161,A -85,B 0,C 180,E1 -11040.783,E2 -11040.783} C_VEL
LIN {X 0,Y 402.962,Z 464.77,A -85,B 0,C 180,E1 -11041.908,E2 -11041.908} C_VEL
LIN {X 0,Y 402.808,Z 466.834,A -85,B 0,C 180,E1 -11043.024,E2 -11043.024} C_VEL
LIN {X 0,Y 402.699,Z 468.317,A -85,B 0,C 180,E1 -11044.133,E2 -11044.133} C_VEL
LIN {X 0,Y 402.636,Z 469.331,A -85,B 0,C 180,E1 -11045.235,E2 -11045.235} C_VEL
LIN {X 0,Y 402.597,Z 469.841,A -85,B 0,C 180,E1 -11046.329,E2 -11046.329} C_VEL
LIN {X 0,Y 402.596,Z 469.824,A -85,B 0,C 180,E1 -11047.686,E2 -11047.686} C_VEL
LIN {X 0,Y 402.674,Z 468.565,A -85,B 0,C 180,E1 -11049.571,E2 -11049.571} C_VEL
LIN {X 0,Y 402.786,Z 467.208,A -85,B 0,C 180,E1 -11050.64,E2 -11050.64} C_VEL
LIN {X 0,Y 402.951,Z 464.314,A -85,B 0,C 180,E1 -11052.229,E2 -11052.229} C_VEL
LIN {X 0,Y 403.186,Z 460.316,A -85,B 0,C 180,E1 -11053.807,E2 -11053.807} C_VEL
LIN {X 0,Y 403.544,Z 455.113,A -85,B 0,C 180,E1 -11055.374,E2 -11055.374} C_VEL
LIN {X 0,Y 404.034,Z 448.536,A -85,B 0,C 180,E1 -11056.932,E2 -11056.932} C_VEL
LIN {X 0,Y 404.641,Z 440.295,A -85,B 0,C 180,E1 -11058.479,E2 -11058.479} C_VEL
LIN {X 0,Y 405.295,Z 431.875,A -85,B 0,C 180,E1 -11059.763,E2 -11059.763} C_VEL
LIN {X 0,Y 406.122,Z 421.534,A -85,B 0,C 180,E1 -11061.041,E2 -11061.041} C_VEL
LIN {X 0,Y 406.898,Z 411.224,A -85,B 0,C 180,E1 -11062.059,E2 -11062.059} C_VEL
LIN {X 0,Y 407.676,Z 399.948,A -85,B 0,C 180,E1 -11062.945,E2 -11062.945} C_VEL
LIN {X 0,Y 408.285,Z 387.509,A -85,B 0,C 180,E1 -11063.701,E2 -11063.701} C_VEL
LIN {X 0,Y 408.871,Z 374.429,A -85,B 0,C 180,E1 -11064.255,E2 -11064.255} C_VEL
LIN {X 0,Y 408.662,Z 368.708,A -85,B 0,C 180,E1 -11064.452,E2 -11064.452} C_VEL
LIN {X 0,Y 406.097,Z 359.421,A -85,B 0,C 180,E1 -11064.78,E2 -11064.78} C_VEL
LIN {X 0,Y 403.333,Z 350.079,A -85,B 0,C 180,E1 -11065.075,E2 -11065.075} C_VEL
LIN {X 0,Y 402.699,Z 344.257,A -85,B 0,C 180,E1 -11065.208,E2 -11065.208} C_VEL
LIN {X 0,Y 403.457,Z 282.291,A -85,B 0,C 180,E1 -11066.332,E2 -11066.332} C_VEL
LIN {X 0,Y 399.159,Z 259.085,A -85,B 0,C 180,E1 -11067.005,E2 -11067.005} C_VEL
LIN {X 0,Y 399.624,Z 250.439,A -85,B 0,C 180,E1 -11068.993,E2 -11068.993} C_VEL
LIN {X 0,Y 398.333,Z 242.457,A -85,B 0,C 180,E1 -11071.012,E2 -11071.012} C_VEL
LIN {X 0,Y 397.394,Z 237.542,A -85,B 0,C 180,E1 -11072.345,E2 -11072.345} C_VEL
LIN {X 0,Y 397.337,Z 237.489,A -85,B 0,C 180,E1 -11076.093,E2 -11076.093} C_VEL
LIN {X 0,Y 397.218,Z 237.503,A -85,B 0,C 180,E1 -11079.163,E2 -11079.163} C_VEL
LIN {X 0,Y 397.194,Z 237.5,A -85,B 0,C 180,E1 -11082.26,E2 -11082.26} C_VEL
LIN {X 0,Y 397.145,Z 237.515,A -85,B 0,C 180,E1 -11085.394,E2 -11085.394} C_VEL
LIN {X 0,Y 397.128,Z 237.514,A -85,B 0,C 180,E1 -11088.576,E2 -11088.576} C_VEL
LIN {X 0,Y 397.063,Z 237.526,A -85,B 0,C 180,E1 -11091.821,E2 -11091.821} C_VEL
LIN {X 0,Y 397.092,Z 237.516,A -85,B 0,C 180,E1 -11095.137,E2 -11095.137} C_VEL
LIN {X 0,Y 397.048,Z 237.518,A -85,B 0,C 180,E1 -11098.55,E2 -11098.55} C_VEL
LIN {X 0,Y 397.052,Z 237.525,A -85,B 0,C 180,E1 -11101.839,E2 -11101.839} C_VEL
LIN {X 0,Y 397.089,Z 237.512,A -85,B 0,C 180,E1 -11104.498,E2 -11104.498} C_VEL
LIN {X 0,Y 397.064,Z 237.525,A -85,B 0,C 180,E1 -11108.28,E2 -11108.28} C_VEL
LIN {X 0,Y 397.027,Z 237.518,A -85,B 0,C 180,E1 -11111.98,E2 -11111.98} C_VEL
LIN {X 0,Y 397.063,Z 237.524,A -85,B 0,C 180,E1 -11115.073,E2 -11115.073} C_VEL
LIN {X 0,Y 397.031,Z 237.525,A -85,B 0,C 180,E1 -11118.028,E2 -11118.028} C_VEL
LIN {X 0,Y 397.074,Z 237.505,A -85,B 0,C 180,E1 -11121.728,E2 -11121.728} C_VEL
LIN {X 0,Y 397.101,Z 237.519,A -85,B 0,C 180,E1 -11125.51,E2 -11125.51} C_VEL
LIN {X 0,Y 397.062,Z 237.515,A -85,B 0,C 180,E1 -11129.121,E2 -11129.121} C_VEL
LIN {X 0,Y 397.048,Z 237.506,A -85,B 0,C 180,E1 -11132.256,E2 -11132.256} C_VEL
LIN {X 0,Y 397.092,Z 237.514,A -85,B 0,C 180,E1 -11134.869,E2 -11134.869} C_VEL
LIN {X 0,Y 397.086,Z 237.516,A -85,B 0,C 180,E1 -11138.185,E2 -11138.185} C_VEL
LIN {X 0,Y 397.15,Z 237.493,A -85,B 0,C 180,E1 -11141.43,E2 -11141.43} C_VEL
LIN {X 0,Y 397.173,Z 237.497,A -85,B 0,C 180,E1 -11144.612,E2 -11144.612} C_VEL
LIN {X 0,Y 397.211,Z 237.508,A -85,B 0,C 180,E1 -11147.746,E2 -11147.746} C_VEL
LIN {X 0,Y 397.227,Z 237.495,A -85,B 0,C 180,E1 -11150.841,E2 -11150.841} C_VEL
LIN {X 0,Y 397.32,Z 237.469,A -85,B 0,C 180,E1 -11153.911,E2 -11153.911} C_VEL
LIN {X 0,Y 397.441,Z 237.473,A -85,B 0,C 180,E1 -11157.977,E2 -11157.977} C_VEL
LIN {X 0,Y 397.44,Z 237.475,A -85,B 0,C 180,E1 -11162.03,E2 -11162.03} C_VEL
LIN {X 0,Y 397.349,Z 237.467,A -85,B 0,C 180,E1 -11166.095,E2 -11166.095} C_VEL
LIN {X 0,Y 397.238,Z 237.5,A -85,B 0,C 180,E1 -11169.165,E2 -11169.165} C_VEL
LIN {X 0,Y 397.225,Z 237.504,A -85,B 0,C 180,E1 -11172.261,E2 -11172.261} C_VEL
LIN {X 0,Y 397.185,Z 237.49,A -85,B 0,C 180,E1 -11175.395,E2 -11175.395} C_VEL
LIN {X 0,Y 397.166,Z 237.509,A -85,B 0,C 180,E1 -11178.576,E2 -11178.576} C_VEL
LIN {X 0,Y 397.105,Z 237.513,A -85,B 0,C 180,E1 -11181.821,E2 -11181.821} C_VEL
LIN {X 0,Y 397.117,Z 237.508,A -85,B 0,C 180,E1 -11185.137,E2 -11185.137} C_VEL
LIN {X 0,Y 397.082,Z 237.521,A -85,B 0,C 180,E1 -11188.55,E2 -11188.55} C_VEL
LIN {X 0,Y 397.091,Z 237.513,A -85,B 0,C 180,E1 -11191.838,E2 -11191.838} C_VEL
LIN {X 0,Y 397.13,Z 237.514,A -85,B 0,C 180,E1 -11194.496,E2 -11194.496} C_VEL
LIN {X 0,Y 397.103,Z 237.513,A -85,B 0,C 180,E1 -11198.278,E2 -11198.278} C_VEL
LIN {X 0,Y 397.065,Z 237.517,A -85,B 0,C 180,E1 -11201.978,E2 -11201.978} C_VEL
LIN {X 0,Y 397.096,Z 237.52,A -85,B 0,C 180,E1 -11205.07,E2 -11205.07} C_VEL
LIN {X 0,Y 397.065,Z 237.525,A -85,B 0,C 180,E1 -11208.024,E2 -11208.024} C_VEL
LIN {X 0,Y 397.103,Z 237.521,A -85,B 0,C 180,E1 -11211.724,E2 -11211.724} C_VEL
LIN {X 0,Y 397.137,Z 237.517,A -85,B 0,C 180,E1 -11215.507,E2 -11215.507} C_VEL
LIN {X 0,Y 397.09,Z 237.518,A -85,B 0,C 180,E1 -11219.118,E2 -11219.118} C_VEL
LIN {X 0,Y 397.176,Z 237.586,A -85,B 0,C 180,E1 -11222.679,E2 -11222.679} C_VEL
LIN {X 0,Y 398.67,Z 245.016,A -85,B 0,C 180,E1 -11224.568,E2 -11224.568} C_VEL
LIN {X 0,Y 400.106,Z 252.825,A -85,B 0,C 180,E1 -11226.445,E2 -11226.445} C_VEL
LIN {X 0,Y 399.202,Z 266.094,A -85,B 0,C 180,E1 -11229.383,E2 -11229.383} C_VEL
LIN {X 0,Y 399.027,Z 269.39,A -85,B 0,C 180,E1 -11230.034,E2 -11230.034} C_VEL
LIN {X 0,Y 403.372,Z 295.357,A -85,B 0,C 180,E1 -11230.753,E2 -11230.753} C_VEL
LIN {X 0,Y 402.318,Z 377.424,A -85,B 0,C 180,E1 -11232.264,E2 -11232.264} C_VEL
LIN {X 0,Y 401.711,Z 391.23,A -85,B 0,C 180,E1 -11232.73,E2 -11232.73} C_VEL
LIN {X 0,Y 401.04,Z 404.151,A -85,B 0,C 180,E1 -11233.389,E2 -11233.389} C_VEL
LIN {X 0,Y 400.23,Z 415.922,A -85,B 0,C 180,E1 -11234.205,E2 -11234.205} C_VEL
LIN {X 0,Y 399.361,Z 427.795,A -85,B 0,C 180,E1 -11235.268,E2 -11235.268} C_VEL
LIN {X 0,Y 398.539,Z 438.502,A -85,B 0,C 180,E1 -11236.488,E2 -11236.488} C_VEL
LIN {X 0,Y 397.774,Z 447.515,A -85,B 0,C 180,E1 -11237.759,E2 -11237.759} C_VEL
LIN {X 0,Y 397.038,Z 456.326,A -85,B 0,C 180,E1 -11239.288,E2 -11239.288} C_VEL
LIN {X 0,Y 396.536,Z 463.358,A -85,B 0,C 180,E1 -11240.821,E2 -11240.821} C_VEL
LIN {X 0,Y 396.162,Z 468.98,A -85,B 0,C 180,E1 -11242.353,E2 -11242.353} C_VEL
LIN {X 0,Y 395.867,Z 474.047,A -85,B 0,C 180,E1 -11244.151,E2 -11244.151} C_VEL
LIN {X 0,Y 395.771,Z 477.63,A -85,B 0,C 180,E1 -11245.926,E2 -11245.926} C_VEL
LIN {X 0,Y 395.695,Z 479.079,A -85,B 0,C 180,E1 -11246.945,E2 -11246.945} C_VEL
LIN {X 0,Y 395.723,Z 480.102,A -85,B 0,C 180,E1 -11247.964,E2 -11247.964} C_VEL
LIN {X 0,Y 395.761,Z 480.737,A -85,B 0,C 180,E1 -11248.982,E2 -11248.982} C_VEL
LIN {X 0,Y 395.764,Z 480.984,A -85,B 0,C 180,E1 -11249.999,E2 -11249.999} C_VEL
LIN {X 0,Y 395.76,Z 480.81,A -85,B 0,C 180,E1 -11251.017,E2 -11251.017} C_VEL
LIN {X 0,Y 395.723,Z 480.224,A -85,B 0,C 180,E1 -11252.035,E2 -11252.035} C_VEL
LIN {X 0,Y 395.775,Z 477.881,A -85,B 0,C 180,E1 -11254.072,E2 -11254.072} C_VEL
LIN {X 0,Y 395.876,Z 474.986,A -85,B 0,C 180,E1 -11255.602,E2 -11255.602} C_VEL
LIN {X 0,Y 396.061,Z 471.061,A -85,B 0,C 180,E1 -11257.134,E2 -11257.134} C_VEL
LIN {X 0,Y 396.401,Z 466.007,A -85,B 0,C 180,E1 -11258.667,E2 -11258.667} C_VEL
LIN {X 0,Y 396.886,Z 459.659,A -85,B 0,C 180,E1 -11260.199,E2 -11260.199} C_VEL
LIN {X 0,Y 397.541,Z 451.713,A -85,B 0,C 180,E1 -11261.729,E2 -11261.729} C_VEL
LIN {X 0,Y 398.514,Z 441.84,A -85,B 0,C 180,E1 -11263.253,E2 -11263.253} C_VEL
LIN {X 0,Y 399.308,Z 431.533,A -85,B 0,C 180,E1 -11264.522,E2 -11264.522} C_VEL
LIN {X 0,Y 400.164,Z 421.302,A -85,B 0,C 180,E1 -11265.534,E2 -11265.534} C_VEL
LIN {X 0,Y 400.988,Z 410.152,A -85,B 0,C 180,E1 -11266.416,E2 -11266.416} C_VEL
LIN {X 0,Y 401.785,Z 397.709,A -85,B 0,C 180,E1 -11267.167,E2 -11267.167} C_VEL
LIN {X 0,Y 402.451,Z 384.444,A -85,B 0,C 180,E1 -11267.728,E2 -11267.728} C_VEL
LIN {X 0,Y 402.891,Z 371.58,A -85,B 0,C 180,E1 -11268.069,E2 -11268.069} C_VEL
LIN {X 0,Y 403.895,Z 295.759,A -85,B 0,C 180,E1 -11269.453,E2 -11269.453} C_VEL
LIN {X 0,Y 399.808,Z 272.247,A -85,B 0,C 180,E1 -11270.123,E2 -11270.123} C_VEL
LIN {X 0,Y 399.186,Z 268.945,A -85,B 0,C 180,E1 -11270.252,E2 -11270.252} C_VEL
LIN {X 0,Y 400.26,Z 254.796,A -85,B 0,C 180,E1 -11273.269,E2 -11273.269} C_VEL
LIN {X 0,Y 399.662,Z 249.901,A -85,B 0,C 180,E1 -11274.407,E2 -11274.407} C_VEL
LIN {X 0,Y 397.473,Z 238.91,A -85,B 0,C 180,E1 -11277.083,E2 -11277.083} C_VEL
LIN {X 0,Y 397.204,Z 237.531,A -85,B 0,C 180,E1 -11277.531,E2 -11277.531} C_VEL
LIN {X 0,Y 397.084,Z 237.523,A -85,B 0,C 180,E1 -11280.881,E2 -11280.881} C_VEL
LIN {X 0,Y 397.13,Z 237.517,A -85,B 0,C 180,E1 -11284.491,E2 -11284.491} C_VEL
LIN {X 0,Y 397.096,Z 237.523,A -85,B 0,C 180,E1 -11288.274,E2 -11288.274} C_VEL
LIN {X 0,Y 397.062,Z 237.526,A -85,B 0,C 180,E1 -11291.975,E2 -11291.975} C_VEL
LIN {X 0,Y 397.089,Z 237.519,A -85,B 0,C 180,E1 -11295.067,E2 -11295.067} C_VEL
LIN {X 0,Y 397.061,Z 237.526,A -85,B 0,C 180,E1 -11298.02,E2 -11298.02} C_VEL
LIN {X 0,Y 397.094,Z 237.515,A -85,B 0,C 180,E1 -11301.721,E2 -11301.721} C_VEL
LIN {X 0,Y 397.118,Z 237.513,A -85,B 0,C 180,E1 -11305.503,E2 -11305.503} C_VEL
LIN {X 0,Y 397.078,Z 237.521,A -85,B 0,C 180,E1 -11309.115,E2 -11309.115} C_VEL
LIN {X 0,Y 397.063,Z 237.522,A -85,B 0,C 180,E1 -11312.249,E2 -11312.249} C_VEL
LIN {X 0,Y 397.102,Z 237.523,A -85,B 0,C 180,E1 -11314.862,E2 -11314.862} C_VEL
LIN {X 0,Y 397.093,Z 237.515,A -85,B 0,C 180,E1 -11318.178,E2 -11318.178} C_VEL
LIN {X 0,Y 397.155,Z 237.505,A -85,B 0,C 180,E1 -11321.423,E2 -11321.423} C_VEL
LIN {X 0,Y 397.173,Z 237.51,A -85,B 0,C 180,E1 -11324.605,E2 -11324.605} C_VEL
LIN {X 0,Y 397.213,Z 237.504,A -85,B 0,C 180,E1 -11327.739,E2 -11327.739} C_VEL
LIN {X 0,Y 397.223,Z 237.502,A -85,B 0,C 180,E1 -11330.834,E2 -11330.834} C_VEL
LIN {X 0,Y 397.34,Z 237.489,A -85,B 0,C 180,E1 -11333.905,E2 -11333.905} C_VEL
LIN {X 0,Y 397.427,Z 237.479,A -85,B 0,C 180,E1 -11337.97,E2 -11337.97} C_VEL
LIN {X 0,Y 397.425,Z 237.479,A -85,B 0,C 180,E1 -11342.023,E2 -11342.023} C_VEL
LIN {X 0,Y 397.278,Z 237.493,A -85,B 0,C 180,E1 -11346.468,E2 -11346.468} C_VEL
LIN {X 0,Y 397.213,Z 237.503,A -85,B 0,C 180,E1 -11349.159,E2 -11349.159} C_VEL
LIN {X 0,Y 397.199,Z 237.507,A -85,B 0,C 180,E1 -11352.255,E2 -11352.255} C_VEL
LIN {X 0,Y 397.161,Z 237.512,A -85,B 0,C 180,E1 -11355.389,E2 -11355.389} C_VEL
LIN {X 0,Y 397.139,Z 237.516,A -85,B 0,C 180,E1 -11358.57,E2 -11358.57} C_VEL
LIN {X 0,Y 397.077,Z 237.524,A -85,B 0,C 180,E1 -11361.815,E2 -11361.815} C_VEL
LIN {X 0,Y 397.102,Z 237.516,A -85,B 0,C 180,E1 -11365.131,E2 -11365.131} C_VEL
LIN {X 0,Y 397.056,Z 237.519,A -85,B 0,C 180,E1 -11368.544,E2 -11368.544} C_VEL
LIN {X 0,Y 397.058,Z 237.522,A -85,B 0,C 180,E1 -11371.833,E2 -11371.833} C_VEL
LIN {X 0,Y 397.101,Z 237.519,A -85,B 0,C 180,E1 -11374.49,E2 -11374.49} C_VEL
LIN {X 0,Y 397.083,Z 237.523,A -85,B 0,C 180,E1 -11378.271,E2 -11378.271} C_VEL
LIN {X 0,Y 397.147,Z 237.665,A -85,B 0,C 180,E1 -11381.826,E2 -11381.826} C_VEL
LIN {X 0,Y 399.513,Z 249.293,A -85,B 0,C 180,E1 -11384.714,E2 -11384.714} C_VEL
LIN {X 0,Y 399.702,Z 253.993,A -85,B 0,C 180,E1 -11385.791,E2 -11385.791} C_VEL
LIN {X 0,Y 399.448,Z 258.886,A -85,B 0,C 180,E1 -11386.803,E2 -11386.803} C_VEL
LIN {X 0,Y 402.128,Z 272.24,A -85,B 0,C 180,E1 -11387.246,E2 -11387.246} C_VEL
LIN {X 0,Y 404.046,Z 282.636,A -85,B 0,C 180,E1 -11387.547,E2 -11387.547} C_VEL
LIN {X 0,Y 402.759,Z 366.326,A -85,B 0,C 180,E1 -11389.089,E2 -11389.089} C_VEL
LIN {X 0,Y 402.257,Z 379.861,A -85,B 0,C 180,E1 -11389.543,E2 -11389.543} C_VEL
LIN {X 0,Y 401.666,Z 392.676,A -85,B 0,C 180,E1 -11390.188,E2 -11390.188} C_VEL
LIN {X 0,Y 400.891,Z 404.886,A -85,B 0,C 180,E1 -11391.031,E2 -11391.031} C_VEL
LIN {X 0,Y 399.961,Z 416.344,A -85,B 0,C 180,E1 -11392.049,E2 -11392.049} C_VEL
LIN {X 0,Y 399.045,Z 426.792,A -85,B 0,C 180,E1 -11393.217,E2 -11393.217} C_VEL
LIN {X 0,Y 398.344,Z 435.317,A -85,B 0,C 180,E1 -11394.395,E2 -11394.395} C_VEL
LIN {X 0,Y 397.525,Z 444.376,A -85,B 0,C 180,E1 -11395.935,E2 -11395.935} C_VEL
LIN {X 0,Y 396.838,Z 452.21,A -85,B 0,C 180,E1 -11397.608,E2 -11397.608} C_VEL
LIN {X 0,Y 396.416,Z 457.6,A -85,B 0,C 180,E1 -11399.061,E2 -11399.061} C_VEL
LIN {X 0,Y 396.04,Z 462.77,A -85,B 0,C 180,E1 -11400.869,E2 -11400.869} C_VEL
LIN {X 0,Y 395.774,Z 466.35,A -85,B 0,C 180,E1 -11402.597,E2 -11402.597} C_VEL
LIN {X 0,Y 395.634,Z 467.921,A -85,B 0,C 180,E1 -11403.636,E2 -11403.636} C_VEL
LIN {X 0,Y 395.567,Z 469.251,A -85,B 0,C 180,E1 -11404.961,E2 -11404.961} C_VEL
LIN {X 0,Y 395.494,Z 470.032,A -85,B 0,C 180,E1 -11406.988,E2 -11406.988} C_VEL
LIN {X 0,Y 395.496,Z 469.76,A -85,B 0,C 180,E1 -11408.09,E2 -11408.09} C_VEL
LIN {X 0,Y 395.538,Z 469.054,A -85,B 0,C 180,E1 -11409.185,E2 -11409.185} C_VEL
LIN {X 0,Y 395.659,Z 467.898,A -85,B 0,C 180,E1 -11410.277,E2 -11410.277} C_VEL
LIN {X 0,Y 395.841,Z 465.269,A -85,B 0,C 180,E1 -11411.899,E2 -11411.899} C_VEL
LIN {X 0,Y 396.038,Z 461.556,A -85,B 0,C 180,E1 -11413.506,E2 -11413.506} C_VEL
LIN {X 0,Y 396.369,Z 456.655,A -85,B 0,C 180,E1 -11415.103,E2 -11415.103} C_VEL
LIN {X 0,Y 396.903,Z 449.715,A -85,B 0,C 180,E1 -11416.855,E2 -11416.855} C_VEL
LIN {X 0,Y 397.444,Z 442.691,A -85,B 0,C 180,E1 -11418.268,E2 -11418.268} C_VEL
LIN {X 0,Y 398.153,Z 434.735,A -85,B 0,C 180,E1 -11419.577,E2 -11419.577} C_VEL
LIN {X 0,Y 398.948,Z 424.997,A -85,B 0,C 180,E1 -11420.878,E2 -11420.878} C_VEL
LIN {X 0,Y 399.835,Z 414.137,A -85,B 0,C 180,E1 -11422.044,E2 -11422.044} C_VEL
LIN {X 0,Y 400.628,Z 403.613,A -85,B 0,C 180,E1 -11422.947,E2 -11422.947} C_VEL
LIN {X 0,Y 401.312,Z 391.094,A -85,B 0,C 180,E1 -11423.78,E2 -11423.78} C_VEL
LIN {X 0,Y 401.927,Z 377.905,A -85,B 0,C 180,E1 -11424.415,E2 -11424.415} C_VEL
LIN {X 0,Y 402.355,Z 365.439,A -85,B 0,C 180,E1 -11424.811,E2 -11424.811} C_VEL
LIN {X 0,Y 402.699,Z 344.257,A -85,B 0,C 180,E1 -11425.208,E2 -11425.208} C_VEL
LIN {X 0,Y 402.09,Z 338.445,A -85,B 0,C 180,E1 -11425.343,E2 -11425.343} C_VEL
LIN {X 0,Y 396.788,Z 319.76,A -85,B 0,C 180,E1 -11425.938,E2 -11425.938} C_VEL
LIN {X 0,Y 396.325,Z 313.948,A -85,B 0,C 180,E1 -11426.07,E2 -11426.07} C_VEL
LIN {X 0,Y 396.733,Z 283.235,A -85,B 0,C 180,E1 -11426.639,E2 -11426.639} C_VEL
LIN {X 0,Y 392.266,Z 259.059,A -85,B 0,C 180,E1 -11427.363,E2 -11427.363} C_VEL
LIN {X 0,Y 392.69,Z 252.178,A -85,B 0,C 180,E1 -11428.975,E2 -11428.975} C_VEL
LIN {X 0,Y 391.447,Z 244.18,A -85,B 0,C 180,E1 -11431.03,E2 -11431.03} C_VEL
LIN {X 0,Y 390.342,Z 238.419,A -85,B 0,C 180,E1 -11432.613,E2 -11432.613} C_VEL
LIN {X 0,Y 390.291,Z 238.367,A -85,B 0,C 180,E1 -11436.203,E2 -11436.203} C_VEL
LIN {X 0,Y 390.171,Z 238.38,A -85,B 0,C 180,E1 -11439.33,E2 -11439.33} C_VEL
LIN {X 0,Y 390.143,Z 238.377,A -85,B 0,C 180,E1 -11442.485,E2 -11442.485} C_VEL
LIN {X 0,Y 390.105,Z 238.392,A -85,B 0,C 180,E1 -11445.679,E2 -11445.679} C_VEL
LIN {X 0,Y 390.072,Z 238.392,A -85,B 0,C 180,E1 -11448.924,E2 -11448.924} C_VEL
LIN {X 0,Y 390.005,Z 238.405,A -85,B 0,C 180,E1 -11452.237,E2 -11452.237} C_VEL
LIN {X 0,Y 390.037,Z 238.397,A -85,B 0,C 180,E1 -11455.73,E2 -11455.73} C_VEL
LIN {X 0,Y 390.003,Z 238.392,A -85,B 0,C 180,E1 -11459.115,E2 -11459.115} C_VEL
LIN {X 0,Y 390.013,Z 238.401,A -85,B 0,C 180,E1 -11462.725,E2 -11462.725} C_VEL
LIN {X 0,Y 390.015,Z 238.389,A -85,B 0,C 180,E1 -11465.826,E2 -11465.826} C_VEL
LIN {X 0,Y 390.01,Z 238.401,A -85,B 0,C 180,E1 -11469.216,E2 -11469.216} C_VEL
LIN {X 0,Y 390.006,Z 238.391,A -85,B 0,C 180,E1 -11472.376,E2 -11472.376} C_VEL
LIN {X 0,Y 390.019,Z 238.399,A -85,B 0,C 180,E1 -11475.358,E2 -11475.358} C_VEL
LIN {X 0,Y 389.994,Z 238.402,A -85,B 0,C 180,E1 -11478.188,E2 -11478.188} C_VEL
LIN {X 0,Y 390.039,Z 238.382,A -85,B 0,C 180,E1 -11480.908,E2 -11480.908} C_VEL
LIN {X 0,Y 390.053,Z 238.395,A -85,B 0,C 180,E1 -11484.795,E2 -11484.795} C_VEL
LIN {X 0,Y 390.007,Z 238.397,A -85,B 0,C 180,E1 -11488.499,E2 -11488.499} C_VEL
LIN {X 0,Y 390.003,Z 238.384,A -85,B 0,C 180,E1 -11492.007,E2 -11492.007} C_VEL
LIN {X 0,Y 390.033,Z 238.402,A -85,B 0,C 180,E1 -11495.521,E2 -11495.521} C_VEL
LIN {X 0,Y 390.047,Z 238.394,A -85,B 0,C 180,E1 -11498.882,E2 -11498.882} C_VEL
LIN {X 0,Y 390.105,Z 238.362,A -85,B 0,C 180,E1 -11502.17,E2 -11502.17} C_VEL
LIN {X 0,Y 390.139,Z 238.376,A -85,B 0,C 180,E1 -11505.397,E2 -11505.397} C_VEL
LIN {X 0,Y 390.134,Z 238.384,A -85,B 0,C 180,E1 -11508.575,E2 -11508.575} C_VEL
LIN {X 0,Y 390.255,Z 238.356,A -85,B 0,C 180,E1 -11512.09,E2 -11512.09} C_VEL
LIN {X 0,Y 390.2,Z 238.356,A -85,B 0,C 180,E1 -11514.837,E2 -11514.837} C_VEL
LIN {X 0,Y 390.409,Z 238.348,A -85,B 0,C 180,E1 -11517.94,E2 -11517.94} C_VEL
LIN {X 0,Y 390.406,Z 238.35,A -85,B 0,C 180,E1 -11522.067,E2 -11522.067} C_VEL
LIN {X 0,Y 390.305,Z 238.345,A -85,B 0,C 180,E1 -11526.206,E2 -11526.206} C_VEL
LIN {X 0,Y 390.196,Z 238.376,A -85,B 0,C 180,E1 -11529.332,E2 -11529.332} C_VEL
LIN {X 0,Y 390.177,Z 238.38,A -85,B 0,C 180,E1 -11532.486,E2 -11532.486} C_VEL
LIN {X 0,Y 390.146,Z 238.366,A -85,B 0,C 180,E1 -11535.68,E2 -11535.68} C_VEL
LIN {X 0,Y 390.111,Z 238.393,A -85,B 0,C 180,E1 -11538.925,E2 -11538.925} C_VEL
LIN {X 0,Y 390.046,Z 238.393,A -85,B 0,C 180,E1 -11542.237,E2 -11542.237} C_VEL
LIN {X 0,Y 390.06,Z 238.391,A -85,B 0,C 180,E1 -11545.724,E2 -11545.724} C_VEL
LIN {X 0,Y 390.04,Z 238.399,A -85,B 0,C 180,E1 -11549.114,E2 -11549.114} C_VEL
LIN {X 0,Y 390.052,Z 238.39,A -85,B 0,C 180,E1 -11552.724,E2 -11552.724} C_VEL
LIN {X 0,Y 390.064,Z 238.392,A -85,B 0,C 180,E1 -11555.826,E2 -11555.826} C_VEL
LIN {X 0,Y 390.048,Z 238.396,A -85,B 0,C 180,E1 -11559.214,E2 -11559.214} C_VEL
LIN {X 0,Y 390.043,Z 238.389,A -85,B 0,C 180,E1 -11562.374,E2 -11562.374} C_VEL
LIN {X 0,Y 390.052,Z 238.4,A -85,B 0,C 180,E1 -11565.355,E2 -11565.355} C_VEL
LIN {X 0,Y 390.028,Z 238.4,A -85,B 0,C 180,E1 -11568.186,E2 -11568.186} C_VEL
LIN {X 0,Y 390.07,Z 238.394,A -85,B 0,C 180,E1 -11570.904,E2 -11570.904} C_VEL
LIN {X 0,Y 390.097,Z 238.392,A -85,B 0,C 180,E1 -11574.794,E2 -11574.794} C_VEL
LIN {X 0,Y 390.035,Z 238.4,A -85,B 0,C 180,E1 -11578.496,E2 -11578.496} C_VEL
LIN {X 0,Y 390.175,Z 238.515,A -85,B 0,C 180,E1 -11582.438,E2 -11582.438} C_VEL
LIN {X 0,Y 392.836,Z 252.057,A -85,B 0,C 180,E1 -11585.845,E2 -11585.845} C_VEL
LIN {X 0,Y 393.179,Z 255.137,A -85,B 0,C 180,E1 -11586.579,E2 -11586.579} C_VEL
LIN {X 0,Y 392.122,Z 269.174,A -85,B 0,C 180,E1 -11589.68,E2 -11589.68} C_VEL
LIN {X 0,Y 396.669,Z 296.426,A -85,B 0,C 180,E1 -11590.454,E2 -11590.454} C_VEL
LIN {X 0,Y 395.556,Z 376.654,A -85,B 0,C 180,E1 -11591.951,E2 -11591.951} C_VEL
LIN {X 0,Y 394.982,Z 389.921,A -85,B 0,C 180,E1 -11592.392,E2 -11592.392} C_VEL
LIN {X 0,Y 394.32,Z 402.668,A -85,B 0,C 180,E1 -11593.03,E2 -11593.03} C_VEL
LIN {X 0,Y 393.516,Z 413.999,A -85,B 0,C 180,E1 -11593.795,E2 -11593.795} C_VEL
LIN {X 0,Y 392.574,Z 426.077,A -85,B 0,C 180,E1 -11594.861,E2 -11594.861} C_VEL
LIN {X 0,Y 391.749,Z 436.667,A -85,B 0,C 180,E1 -11596.041,E2 -11596.041} C_VEL
LIN {X 0,Y 390.971,Z 445.664,A -85,B 0,C 180,E1 -11597.278,E2 -11597.278} C_VEL
LIN {X 0,Y 390.119,Z 454.774,A -85,B 0,C 180,E1 -11598.833,E2 -11598.833} C_VEL
LIN {X 0,Y 389.55,Z 462.115,A -85,B 0,C 180,E1 -11600.393,E2 -11600.393} C_VEL
LIN {X 0,Y 389.208,Z 467.085,A -85,B 0,C 180,E1 -11601.693,E2 -11601.693} C_VEL
LIN {X 0,Y 388.891,Z 471.905,A -85,B 0,C 180,E1 -11603.253,E2 -11603.253} C_VEL
LIN {X 0,Y 388.764,Z 475.6,A -85,B 0,C 180,E1 -11604.813,E2 -11604.813} C_VEL
LIN {X 0,Y 388.698,Z 477.507,A -85,B 0,C 180,E1 -11605.852,E2 -11605.852} C_VEL
LIN {X 0,Y 388.605,Z 478.965,A -85,B 0,C 180,E1 -11606.889,E2 -11606.889} C_VEL
LIN {X 0,Y 388.621,Z 479.993,A -85,B 0,C 180,E1 -11607.926,E2 -11607.926} C_VEL
LIN {X 0,Y 388.659,Z 480.632,A -85,B 0,C 180,E1 -11608.963,E2 -11608.963} C_VEL
LIN {X 0,Y 388.677,Z 480.883,A -85,B 0,C 180,E1 -11609.999,E2 -11609.999} C_VEL
LIN {X 0,Y 388.659,Z 480.718,A -85,B 0,C 180,E1 -11611.035,E2 -11611.035} C_VEL
LIN {X 0,Y 388.605,Z 479.166,A -85,B 0,C 180,E1 -11613.109,E2 -11613.109} C_VEL
LIN {X 0,Y 388.703,Z 477.802,A -85,B 0,C 180,E1 -11614.147,E2 -11614.147} C_VEL
LIN {X 0,Y 388.785,Z 474.675,A -85,B 0,C 180,E1 -11615.821,E2 -11615.821} C_VEL
LIN {X 0,Y 389.011,Z 471.004,A -85,B 0,C 180,E1 -11617.264,E2 -11617.264} C_VEL
LIN {X 0,Y 389.368,Z 465.962,A -85,B 0,C 180,E1 -11618.824,E2 -11618.824} C_VEL
LIN {X 0,Y 389.897,Z 459.629,A -85,B 0,C 180,E1 -11620.384,E2 -11620.384} C_VEL
LIN {X 0,Y 390.568,Z 451.7,A -85,B 0,C 180,E1 -11621.942,E2 -11621.942} C_VEL
LIN {X 0,Y 391.418,Z 443.628,A -85,B 0,C 180,E1 -11623.233,E2 -11623.233} C_VEL
LIN {X 0,Y 392.239,Z 433.788,A -85,B 0,C 180,E1 -11624.527,E2 -11624.527} C_VEL
LIN {X 0,Y 393.043,Z 424.139,A -85,B 0,C 180,E1 -11625.557,E2 -11625.557} C_VEL
LIN {X 0,Y 393.941,Z 413.756,A -85,B 0,C 180,E1 -11626.451,E2 -11626.451} C_VEL
LIN {X 0,Y 394.803,Z 401.298,A -85,B 0,C 180,E1 -11627.28,E2 -11627.28} C_VEL
LIN {X 0,Y 395.556,Z 388.193,A -85,B 0,C 180,E1 -11627.913,E2 -11627.913} C_VEL
LIN {X 0,Y 396.089,Z 375.128,A -85,B 0,C 180,E1 -11628.323,E2 -11628.323} C_VEL
LIN {X 0,Y 397.181,Z 296.349,A -85,B 0,C 180,E1 -11629.8,E2 -11629.8} C_VEL
LIN {X 0,Y 393.142,Z 272.952,A -85,B 0,C 180,E1 -11630.487,E2 -11630.487} C_VEL
LIN {X 0,Y 392.313,Z 268.634,A -85,B 0,C 180,E1 -11630.673,E2 -11630.673} C_VEL
LIN {X 0,Y 393.344,Z 256.034,A -85,B 0,C 180,E1 -11633.419,E2 -11633.419} C_VEL
LIN {X 0,Y 392.472,Z 249.895,A -85,B 0,C 180,E1 -11634.885,E2 -11634.885} C_VEL
LIN {X 0,Y 390.238,Z 238.912,A -85,B 0,C 180,E1 -11637.628,E2 -11637.628} C_VEL
LIN {X 0,Y 390.125,Z 238.395,A -85,B 0,C 180,E1 -11637.928,E2 -11637.928} C_VEL
LIN {X 0,Y 390.029,Z 238.4,A -85,B 0,C 180,E1 -11641.503,E2 -11641.503} C_VEL
LIN {X 0,Y 390.09,Z 238.394,A -85,B 0,C 180,E1 -11645.205,E2 -11645.205} C_VEL
LIN {X 0,Y 390.062,Z 238.394,A -85,B 0,C 180,E1 -11649.094,E2 -11649.094} C_VEL
LIN {X 0,Y 390.04,Z 238.401,A -85,B 0,C 180,E1 -11652.371,E2 -11652.371} C_VEL
LIN {X 0,Y 390.046,Z 238.396,A -85,B 0,C 180,E1 -11655.352,E2 -11655.352} C_VEL
LIN {X 0,Y 390.023,Z 238.401,A -85,B 0,C 180,E1 -11658.183,E2 -11658.183} C_VEL
LIN {X 0,Y 390.06,Z 238.393,A -85,B 0,C 180,E1 -11660.901,E2 -11660.901} C_VEL
LIN {X 0,Y 390.071,Z 238.393,A -85,B 0,C 180,E1 -11664.789,E2 -11664.789} C_VEL
LIN {X 0,Y 390.023,Z 238.398,A -85,B 0,C 180,E1 -11668.493,E2 -11668.493} C_VEL
LIN {X 0,Y 390.015,Z 238.399,A -85,B 0,C 180,E1 -11672,E2 -11672} C_VEL
LIN {X 0,Y 390.041,Z 238.396,A -85,B 0,C 180,E1 -11675.514,E2 -11675.514} C_VEL
LIN {X 0,Y 390.053,Z 238.398,A -85,B 0,C 180,E1 -11678.875,E2 -11678.875} C_VEL
LIN {X 0,Y 390.108,Z 238.381,A -85,B 0,C 180,E1 -11682.163,E2 -11682.163} C_VEL
LIN {X 0,Y 390.138,Z 238.383,A -85,B 0,C 180,E1 -11685.389,E2 -11685.389} C_VEL
LIN {X 0,Y 390.137,Z 238.384,A -85,B 0,C 180,E1 -11688.568,E2 -11688.568} C_VEL
LIN {X 0,Y 390.26,Z 238.366,A -85,B 0,C 180,E1 -11692.073,E2 -11692.073} C_VEL
LIN {X 0,Y 390.199,Z 238.378,A -85,B 0,C 180,E1 -11694.83,E2 -11694.83} C_VEL
LIN {X 0,Y 390.393,Z 238.355,A -85,B 0,C 180,E1 -11697.933,E2 -11697.933} C_VEL
LIN {X 0,Y 390.391,Z 238.355,A -85,B 0,C 180,E1 -11702.06,E2 -11702.06} C_VEL
LIN {X 0,Y 390.239,Z 238.371,A -85,B 0,C 180,E1 -11706.459,E2 -11706.459} C_VEL
LIN {X 0,Y 390.172,Z 238.381,A -85,B 0,C 180,E1 -11709.326,E2 -11709.326} C_VEL
LIN {X 0,Y 390.18,Z 238.379,A -85,B 0,C 180,E1 -11713.435,E2 -11713.435} C_VEL
LIN {X 0,Y 390.112,Z 238.385,A -85,B 0,C 180,E1 -11717.295,E2 -11717.295} C_VEL
LIN {X 0,Y 390.069,Z 238.396,A -85,B 0,C 180,E1 -11720.466,E2 -11720.466} C_VEL
LIN {X 0,Y 390.046,Z 238.395,A -85,B 0,C 180,E1 -11723.349,E2 -11723.349} C_VEL
LIN {X 0,Y 390.034,Z 238.401,A -85,B 0,C 180,E1 -11726.769,E2 -11726.769} C_VEL
LIN {X 0,Y 390.014,Z 238.404,A -85,B 0,C 180,E1 -11730.297,E2 -11730.297} C_VEL
LIN {X 0,Y 390.044,Z 238.401,A -85,B 0,C 180,E1 -11734.021,E2 -11734.021} C_VEL
LIN {X 0,Y 390.021,Z 238.399,A -85,B 0,C 180,E1 -11737.548,E2 -11737.548} C_VEL
LIN {X 0,Y 390.056,Z 238.398,A -85,B 0,C 180,E1 -11740.823,E2 -11740.823} C_VEL
LIN {X 0,Y 390.118,Z 238.589,A -85,B 0,C 180,E1 -11741.527,E2 -11741.527} C_VEL
LIN {X 0,Y 392.632,Z 250.874,A -85,B 0,C 180,E1 -11744.626,E2 -11744.626} C_VEL
LIN {X 0,Y 392.75,Z 255.691,A -85,B 0,C 180,E1 -11745.745,E2 -11745.745} C_VEL
LIN {X 0,Y 392.602,Z 258.953,A -85,B 0,C 180,E1 -11746.41,E2 -11746.41} C_VEL
LIN {X 0,Y 395.953,Z 275.646,A -85,B 0,C 180,E1 -11746.968,E2 -11746.968} C_VEL
LIN {X 0,Y 397.421,Z 284.508,A -85,B 0,C 180,E1 -11747.224,E2 -11747.224} C_VEL
LIN {X 0,Y 396.046,Z 366.895,A -85,B 0,C 180,E1 -11748.773,E2 -11748.773} C_VEL
LIN {X 0,Y 395.508,Z 380.532,A -85,B 0,C 180,E1 -11749.244,E2 -11749.244} C_VEL
LIN {X 0,Y 394.939,Z 392.302,A -85,B 0,C 180,E1 -11749.848,E2 -11749.848} C_VEL
LIN {X 0,Y 394.248,Z 403.045,A -85,B 0,C 180,E1 -11750.577,E2 -11750.577} C_VEL
LIN {X 0,Y 393.407,Z 413.596,A -85,B 0,C 180,E1 -11751.484,E2 -11751.484} C_VEL
LIN {X 0,Y 392.431,Z 424.411,A -85,B 0,C 180,E1 -11752.653,E2 -11752.653} C_VEL
LIN {X 0,Y 391.567,Z 433.477,A -85,B 0,C 180,E1 -11753.861,E2 -11753.861} C_VEL
LIN {X 0,Y 390.832,Z 441.469,A -85,B 0,C 180,E1 -11755.158,E2 -11755.158} C_VEL
LIN {X 0,Y 390.143,Z 449.113,A -85,B 0,C 180,E1 -11756.674,E2 -11756.674} C_VEL
LIN {X 0,Y 389.493,Z 456.153,A -85,B 0,C 180,E1 -11758.449,E2 -11758.449} C_VEL
LIN {X 0,Y 389.109,Z 461.232,A -85,B 0,C 180,E1 -11760.097,E2 -11760.097} C_VEL
LIN {X 0,Y 388.782,Z 465.525,A -85,B 0,C 180,E1 -11761.967,E2 -11761.967} C_VEL
LIN {X 0,Y 388.614,Z 467.412,A -85,B 0,C 180,E1 -11763.121,E2 -11763.121} C_VEL
LIN {X 0,Y 388.48,Z 469.229,A -85,B 0,C 180,E1 -11764.751,E2 -11764.751} C_VEL
LIN {X 0,Y 388.394,Z 470.078,A -85,B 0,C 180,E1 -11766.542,E2 -11766.542} C_VEL
LIN {X 0,Y 388.423,Z 470.022,A -85,B 0,C 180,E1 -11767.669,E2 -11767.669} C_VEL
LIN {X 0,Y 388.408,Z 469.482,A -85,B 0,C 180,E1 -11768.785,E2 -11768.785} C_VEL
LIN {X 0,Y 388.558,Z 468.224,A -85,B 0,C 180,E1 -11770.127,E2 -11770.127} C_VEL
LIN {X 0,Y 388.78,Z 465.095,A -85,B 0,C 180,E1 -11772.104,E2 -11772.104} C_VEL
LIN {X 0,Y 388.995,Z 461.189,A -85,B 0,C 180,E1 -11773.776,E2 -11773.776} C_VEL
LIN {X 0,Y 389.347,Z 456.298,A -85,B 0,C 180,E1 -11775.363,E2 -11775.363} C_VEL
LIN {X 0,Y 389.94,Z 449.213,A -85,B 0,C 180,E1 -11777.153,E2 -11777.153} C_VEL
LIN {X 0,Y 390.523,Z 442.081,A -85,B 0,C 180,E1 -11778.583,E2 -11778.583} C_VEL
LIN {X 0,Y 391.338,Z 432.767,A -85,B 0,C 180,E1 -11780.086,E2 -11780.086} C_VEL
LIN {X 0,Y 392.2,Z 422.923,A -85,B 0,C 180,E1 -11781.37,E2 -11781.37} C_VEL
LIN {X 0,Y 393.049,Z 412.922,A -85,B 0,C 180,E1 -11782.423,E2 -11782.423} C_VEL
LIN {X 0,Y 393.881,Z 402.002,A -85,B 0,C 180,E1 -11783.341,E2 -11783.341} C_VEL
LIN {X 0,Y 394.595,Z 388.93,A -85,B 0,C 180,E1 -11784.187,E2 -11784.187} C_VEL
LIN {X 0,Y 395.203,Z 376.634,A -85,B 0,C 180,E1 -11784.759,E2 -11784.759} C_VEL
LIN {X 0,Y 395.609,Z 364.148,A -85,B 0,C 180,E1 -11785.136,E2 -11785.136} C_VEL
LIN {X 0,Y 396.325,Z 313.948,A -85,B 0,C 180,E1 -11786.07,E2 -11786.07} C_VEL
LIN {X 0,Y 396.045,Z 308.13,A -85,B 0,C 180,E1 -11786.195,E2 -11786.195} C_VEL
LIN {X 0,Y 394.045,Z 298.68,A -85,B 0,C 180,E1 -11786.473,E2 -11786.473} C_VEL
LIN {X 0,Y 389.919,Z 283.665,A -85,B 0,C 180,E1 -11786.97,E2 -11786.97} C_VEL
LIN {X 0,Y 385.396,Z 259.331,A -85,B 0,C 180,E1 -11787.705,E2 -11787.705} C_VEL
LIN {X 0,Y 385.735,Z 253.918,A -85,B 0,C 180,E1 -11788.957,E2 -11788.957} C_VEL
LIN {X 0,Y 384.988,Z 247.86,A -85,B 0,C 180,E1 -11790.524,E2 -11790.524} C_VEL
LIN {X 0,Y 383.335,Z 239.555,A -85,B 0,C 180,E1 -11792.759,E2 -11792.759} C_VEL
LIN {X 0,Y 383.218,Z 239.249,A -85,B 0,C 180,E1 -11793.155,E2 -11793.155} C_VEL
LIN {X 0,Y 383.247,Z 239.243,A -85,B 0,C 180,E1 -11796.318,E2 -11796.318} C_VEL
LIN {X 0,Y 383.118,Z 239.258,A -85,B 0,C 180,E1 -11799.504,E2 -11799.504} C_VEL
LIN {X 0,Y 383.107,Z 239.253,A -85,B 0,C 180,E1 -11802.718,E2 -11802.718} C_VEL
LIN {X 0,Y 383.046,Z 239.268,A -85,B 0,C 180,E1 -11805.976,E2 -11805.976} C_VEL
LIN {X 0,Y 383.027,Z 239.271,A -85,B 0,C 180,E1 -11809.286,E2 -11809.286} C_VEL
LIN {X 0,Y 382.959,Z 239.279,A -85,B 0,C 180,E1 -11812.669,E2 -11812.669} C_VEL
LIN {X 0,Y 382.972,Z 239.282,A -85,B 0,C 180,E1 -11816.132,E2 -11816.132} C_VEL
LIN {X 0,Y 382.95,Z 239.271,A -85,B 0,C 180,E1 -11819.704,E2 -11819.704} C_VEL
LIN {X 0,Y 382.971,Z 239.275,A -85,B 0,C 180,E1 -11823.405,E2 -11823.405} C_VEL
LIN {X 0,Y 382.995,Z 239.266,A -85,B 0,C 180,E1 -11826.166,E2 -11826.166} C_VEL
LIN {X 0,Y 382.96,Z 239.278,A -85,B 0,C 180,E1 -11829.584,E2 -11829.584} C_VEL
LIN {X 0,Y 382.983,Z 239.265,A -85,B 0,C 180,E1 -11832.782,E2 -11832.782} C_VEL
LIN {X 0,Y 382.968,Z 239.277,A -85,B 0,C 180,E1 -11835.792,E2 -11835.792} C_VEL
LIN {X 0,Y 382.941,Z 239.279,A -85,B 0,C 180,E1 -11838.805,E2 -11838.805} C_VEL
LIN {X 0,Y 382.976,Z 239.26,A -85,B 0,C 180,E1 -11842.102,E2 -11842.102} C_VEL
LIN {X 0,Y 382.995,Z 239.278,A -85,B 0,C 180,E1 -11845.335,E2 -11845.335} C_VEL
LIN {X 0,Y 382.967,Z 239.27,A -85,B 0,C 180,E1 -11849.085,E2 -11849.085} C_VEL
LIN {X 0,Y 382.957,Z 239.262,A -85,B 0,C 180,E1 -11852.695,E2 -11852.695} C_VEL
LIN {X 0,Y 382.998,Z 239.273,A -85,B 0,C 180,E1 -11856.195,E2 -11856.195} C_VEL
LIN {X 0,Y 383.048,Z 239.261,A -85,B 0,C 180,E1 -11859.603,E2 -11859.603} C_VEL
LIN {X 0,Y 383.088,Z 239.235,A -85,B 0,C 180,E1 -11862.935,E2 -11862.935} C_VEL
LIN {X 0,Y 383.122,Z 239.256,A -85,B 0,C 180,E1 -11866.468,E2 -11866.468} C_VEL
LIN {X 0,Y 383.135,Z 239.251,A -85,B 0,C 180,E1 -11870.501,E2 -11870.501} C_VEL
LIN {X 0,Y 383.233,Z 239.223,A -85,B 0,C 180,E1 -11873.687,E2 -11873.687} C_VEL
LIN {X 0,Y 383.375,Z 239.224,A -85,B 0,C 180,E1 -11877.902,E2 -11877.902} C_VEL
LIN {X 0,Y 383.371,Z 239.225,A -85,B 0,C 180,E1 -11882.105,E2 -11882.105} C_VEL
LIN {X 0,Y 383.262,Z 239.223,A -85,B 0,C 180,E1 -11886.32,E2 -11886.32} C_VEL
LIN {X 0,Y 383.146,Z 239.254,A -85,B 0,C 180,E1 -11889.506,E2 -11889.506} C_VEL
LIN {X 0,Y 383.133,Z 239.247,A -85,B 0,C 180,E1 -11893.539,E2 -11893.539} C_VEL
LIN {X 0,Y 383.103,Z 239.257,A -85,B 0,C 180,E1 -11897.072,E2 -11897.072} C_VEL
LIN {X 0,Y 383.038,Z 239.274,A -85,B 0,C 180,E1 -11900.649,E2 -11900.649} C_VEL
LIN {X 0,Y 383.024,Z 239.253,A -85,B 0,C 180,E1 -11903.811,E2 -11903.811} C_VEL
LIN {X 0,Y 382.997,Z 239.278,A -85,B 0,C 180,E1 -11907.31,E2 -11907.31} C_VEL
LIN {X 0,Y 382.992,Z 239.269,A -85,B 0,C 180,E1 -11910.921,E2 -11910.921} C_VEL
LIN {X 0,Y 383.028,Z 239.272,A -85,B 0,C 180,E1 -11914.67,E2 -11914.67} C_VEL
LIN {X 0,Y 383.005,Z 239.27,A -85,B 0,C 180,E1 -11917.904,E2 -11917.904} C_VEL
LIN {X 0,Y 382.973,Z 239.279,A -85,B 0,C 180,E1 -11921.352,E2 -11921.352} C_VEL
LIN {X 0,Y 383.005,Z 239.274,A -85,B 0,C 180,E1 -11924.304,E2 -11924.304} C_VEL
LIN {X 0,Y 383.023,Z 239.27,A -85,B 0,C 180,E1 -11927.241,E2 -11927.241} C_VEL
LIN {X 0,Y 382.997,Z 239.277,A -85,B 0,C 180,E1 -11930.42,E2 -11930.42} C_VEL
LIN {X 0,Y 383.036,Z 239.273,A -85,B 0,C 180,E1 -11934.045,E2 -11934.045} C_VEL
LIN {X 0,Y 382.999,Z 239.276,A -85,B 0,C 180,E1 -11937.579,E2 -11937.579} C_VEL
LIN {X 0,Y 383.003,Z 239.277,A -85,B 0,C 180,E1 -11940.3,E2 -11940.3} C_VEL
LIN {X 0,Y 383.131,Z 239.471,A -85,B 0,C 180,E1 -11942.19,E2 -11942.19} C_VEL
LIN {X 0,Y 385.45,Z 251.241,A -85,B 0,C 180,E1 -11945.205,E2 -11945.205} C_VEL
LIN {X 0,Y 386.239,Z 256.108,A -85,B 0,C 180,E1 -11946.402,E2 -11946.402} C_VEL
LIN {X 0,Y 385.214,Z 269.129,A -85,B 0,C 180,E1 -11949.325,E2 -11949.325} C_VEL
LIN {X 0,Y 389.91,Z 297.035,A -85,B 0,C 180,E1 -11950.134,E2 -11950.134} C_VEL
LIN {X 0,Y 388.759,Z 377.022,A -85,B 0,C 180,E1 -11951.658,E2 -11951.658} C_VEL
LIN {X 0,Y 388.161,Z 390.13,A -85,B 0,C 180,E1 -11952.107,E2 -11952.107} C_VEL
LIN {X 0,Y 387.442,Z 403.347,A -85,B 0,C 180,E1 -11952.788,E2 -11952.788} C_VEL
LIN {X 0,Y 386.559,Z 415.254,A -85,B 0,C 180,E1 -11953.631,E2 -11953.631} C_VEL
LIN {X 0,Y 385.617,Z 426.694,A -85,B 0,C 180,E1 -11954.676,E2 -11954.676} C_VEL
LIN {X 0,Y 384.798,Z 436.777,A -85,B 0,C 180,E1 -11955.83,E2 -11955.83} C_VEL
LIN {X 0,Y 384.031,Z 445.442,A -85,B 0,C 180,E1 -11957.044,E2 -11957.044} C_VEL
LIN {X 0,Y 383.132,Z 454.577,A -85,B 0,C 180,E1 -11958.626,E2 -11958.626} C_VEL
LIN {X 0,Y 382.538,Z 461.936,A -85,B 0,C 180,E1 -11960.215,E2 -11960.215} C_VEL
LIN {X 0,Y 382.032,Z 468.676,A -85,B 0,C 180,E1 -11962.069,E2 -11962.069} C_VEL
LIN {X 0,Y 381.713,Z 473.596,A -85,B 0,C 180,E1 -11963.859,E2 -11963.859} C_VEL
LIN {X 0,Y 381.626,Z 477.379,A -85,B 0,C 180,E1 -11965.775,E2 -11965.775} C_VEL
LIN {X 0,Y 381.52,Z 478.848,A -85,B 0,C 180,E1 -11966.831,E2 -11966.831} C_VEL
LIN {X 0,Y 381.558,Z 480.525,A -85,B 0,C 180,E1 -11968.944,E2 -11968.944} C_VEL
LIN {X 0,Y 381.577,Z 480.782,A -85,B 0,C 180,E1 -11969.999,E2 -11969.999} C_VEL
LIN {X 0,Y 381.558,Z 480.627,A -85,B 0,C 180,E1 -11971.055,E2 -11971.055} C_VEL
LIN {X 0,Y 381.52,Z 479.085,A -85,B 0,C 180,E1 -11973.167,E2 -11973.167} C_VEL
LIN {X 0,Y 381.632,Z 477.726,A -85,B 0,C 180,E1 -11974.223,E2 -11974.223} C_VEL
LIN {X 0,Y 381.744,Z 474.028,A -85,B 0,C 180,E1 -11976.184,E2 -11976.184} C_VEL
LIN {X 0,Y 382.056,Z 469.393,A -85,B 0,C 180,E1 -11977.929,E2 -11977.929} C_VEL
LIN {X 0,Y 382.555,Z 462.932,A -85,B 0,C 180,E1 -11979.783,E2 -11979.783} C_VEL
LIN {X 0,Y 383.18,Z 455.861,A -85,B 0,C 180,E1 -11981.37,E2 -11981.37} C_VEL
LIN {X 0,Y 384.125,Z 447.034,A -85,B 0,C 180,E1 -11982.951,E2 -11982.951} C_VEL
LIN {X 0,Y 385.065,Z 436.992,A -85,B 0,C 180,E1 -11984.401,E2 -11984.401} C_VEL
LIN {X 0,Y 385.949,Z 427.032,A -85,B 0,C 180,E1 -11985.552,E2 -11985.552} C_VEL
LIN {X 0,Y 387.005,Z 415.44,A -85,B 0,C 180,E1 -11986.619,E2 -11986.619} C_VEL
LIN {X 0,Y 387.903,Z 403.682,A -85,B 0,C 180,E1 -11987.461,E2 -11987.461} C_VEL
LIN {X 0,Y 388.757,Z 390.776,A -85,B 0,C 180,E1 -11988.135,E2 -11988.135} C_VEL
LIN {X 0,Y 389.293,Z 378.154,A -85,B 0,C 180,E1 -11988.586,E2 -11988.586} C_VEL
LIN {X 0,Y 389.842,Z 350.416,A -85,B 0,C 180,E1 -11989.144,E2 -11989.144} C_VEL
LIN {X 0,Y 390.52,Z 296.858,A -85,B 0,C 180,E1 -11990.163,E2 -11990.163} C_VEL
LIN {X 0,Y 386.389,Z 273.32,A -85,B 0,C 180,E1 -11990.877,E2 -11990.877} C_VEL
LIN {X 0,Y 385.476,Z 268.578,A -85,B 0,C 180,E1 -11991.076,E2 -11991.076} C_VEL
LIN {X 0,Y 386.452,Z 257.234,A -85,B 0,C 180,E1 -11993.583,E2 -11993.583} C_VEL
LIN {X 0,Y 385.055,Z 248.674,A -85,B 0,C 180,E1 -11995.688,E2 -11995.688} C_VEL
LIN {X 0,Y 383.135,Z 239.631,A -85,B 0,C 180,E1 -11998.022,E2 -11998.022} C_VEL
LIN {X 0,Y 383.059,Z 239.275,A -85,B 0,C 180,E1 -11998.274,E2 -11998.274} C_VEL
LIN {X 0,Y 383.015,Z 239.275,A -85,B 0,C 180,E1 -12002.148,E2 -12002.148} C_VEL
LIN {X 0,Y 383.024,Z 239.275,A -85,B 0,C 180,E1 -12004.666,E2 -12004.666} C_VEL
LIN {X 0,Y 382.998,Z 239.276,A -85,B 0,C 180,E1 -12007.9,E2 -12007.9} C_VEL
LIN {X 0,Y 382.967,Z 239.277,A -85,B 0,C 180,E1 -12011.348,E2 -12011.348} C_VEL
LIN {X 0,Y 382.999,Z 239.28,A -85,B 0,C 180,E1 -12014.301,E2 -12014.301} C_VEL
LIN {X 0,Y 383.014,Z 239.273,A -85,B 0,C 180,E1 -12017.238,E2 -12017.238} C_VEL
LIN {X 0,Y 382.988,Z 239.279,A -85,B 0,C 180,E1 -12020.416,E2 -12020.416} C_VEL
LIN {X 0,Y 383.016,Z 239.274,A -85,B 0,C 180,E1 -12024.041,E2 -12024.041} C_VEL
LIN {X 0,Y 382.986,Z 239.275,A -85,B 0,C 180,E1 -12027.576,E2 -12027.576} C_VEL
LIN {X 0,Y 382.977,Z 239.278,A -85,B 0,C 180,E1 -12030.296,E2 -12030.296} C_VEL
LIN {X 0,Y 383.002,Z 239.272,A -85,B 0,C 180,E1 -12034.042,E2 -12034.042} C_VEL
LIN {X 0,Y 382.988,Z 239.273,A -85,B 0,C 180,E1 -12037.331,E2 -12037.331} C_VEL
LIN {X 0,Y 383.056,Z 239.268,A -85,B 0,C 180,E1 -12040.713,E2 -12040.713} C_VEL
LIN {X 0,Y 383.076,Z 239.265,A -85,B 0,C 180,E1 -12044.023,E2 -12044.023} C_VEL
LIN {X 0,Y 383.131,Z 239.255,A -85,B 0,C 180,E1 -12047.281,E2 -12047.281} C_VEL
LIN {X 0,Y 383.133,Z 239.255,A -85,B 0,C 180,E1 -12050.494,E2 -12050.494} C_VEL
LIN {X 0,Y 383.252,Z 239.246,A -85,B 0,C 180,E1 -12053.68,E2 -12053.68} C_VEL
LIN {X 0,Y 383.358,Z 239.232,A -85,B 0,C 180,E1 -12057.895,E2 -12057.895} C_VEL
LIN {X 0,Y 383.356,Z 239.231,A -85,B 0,C 180,E1 -12062.098,E2 -12062.098} C_VEL
LIN {X 0,Y 383.205,Z 239.248,A -85,B 0,C 180,E1 -12066.447,E2 -12066.447} C_VEL
LIN {X 0,Y 383.123,Z 239.258,A -85,B 0,C 180,E1 -12069.499,E2 -12069.499} C_VEL
LIN {X 0,Y 383.111,Z 239.26,A -85,B 0,C 180,E1 -12073.532,E2 -12073.532} C_VEL
LIN {X 0,Y 383.077,Z 239.26,A -85,B 0,C 180,E1 -12077.066,E2 -12077.066} C_VEL
LIN {X 0,Y 383.011,Z 239.275,A -85,B 0,C 180,E1 -12080.643,E2 -12080.643} C_VEL
LIN {X 0,Y 382.997,Z 239.275,A -85,B 0,C 180,E1 -12083.805,E2 -12083.805} C_VEL
LIN {X 0,Y 382.972,Z 239.278,A -85,B 0,C 180,E1 -12087.303,E2 -12087.303} C_VEL
LIN {X 0,Y 382.959,Z 239.281,A -85,B 0,C 180,E1 -12090.915,E2 -12090.915} C_VEL
LIN {X 0,Y 382.994,Z 239.275,A -85,B 0,C 180,E1 -12094.665,E2 -12094.665} C_VEL
LIN {X 0,Y 382.977,Z 239.278,A -85,B 0,C 180,E1 -12097.901,E2 -12097.901} C_VEL
LIN {X 0,Y 383.02,Z 239.369,A -85,B 0,C 180,E1 -12101.123,E2 -12101.123} C_VEL
LIN {X 0,Y 385.041,Z 248.826,A -85,B 0,C 180,E1 -12103.62,E2 -12103.62} C_VEL
LIN {X 0,Y 385.958,Z 253.934,A -85,B 0,C 180,E1 -12104.895,E2 -12104.895} C_VEL
LIN {X 0,Y 385.759,Z 258.953,A -85,B 0,C 180,E1 -12105.997,E2 -12105.997} C_VEL
LIN {X 0,Y 388.109,Z 270.257,A -85,B 0,C 180,E1 -12106.406,E2 -12106.406} C_VEL
LIN {X 0,Y 390.807,Z 284.781,A -85,B 0,C 180,E1 -12106.855,E2 -12106.855} C_VEL
LIN {X 0,Y 389.372,Z 366.939,A -85,B 0,C 180,E1 -12108.426,E2 -12108.426} C_VEL
LIN {X 0,Y 388.799,Z 380.737,A -85,B 0,C 180,E1 -12108.912,E2 -12108.912} C_VEL
LIN {X 0,Y 388.141,Z 393.471,A -85,B 0,C 180,E1 -12109.587,E2 -12109.587} C_VEL
LIN {X 0,Y 387.334,Z 404.942,A -85,B 0,C 180,E1 -12110.409,E2 -12110.409} C_VEL
LIN {X 0,Y 386.301,Z 416.454,A -85,B 0,C 180,E1 -12111.464,E2 -12111.464} C_VEL
LIN {X 0,Y 385.338,Z 426.891,A -85,B 0,C 180,E1 -12112.67,E2 -12112.67} C_VEL
LIN {X 0,Y 384.482,Z 435.832,A -85,B 0,C 180,E1 -12113.951,E2 -12113.951} C_VEL
LIN {X 0,Y 383.576,Z 444.751,A -85,B 0,C 180,E1 -12115.529,E2 -12115.529} C_VEL
LIN {X 0,Y 382.812,Z 452.191,A -85,B 0,C 180,E1 -12117.171,E2 -12117.171} C_VEL
LIN {X 0,Y 382.256,Z 458.666,A -85,B 0,C 180,E1 -12119.017,E2 -12119.017} C_VEL
LIN {X 0,Y 381.899,Z 463.451,A -85,B 0,C 180,E1 -12120.814,E2 -12120.814} C_VEL
LIN {X 0,Y 381.603,Z 466.865,A -85,B 0,C 180,E1 -12122.587,E2 -12122.587} C_VEL
LIN {X 0,Y 381.404,Z 469.208,A -85,B 0,C 180,E1 -12124.53,E2 -12124.53} C_VEL
LIN {X 0,Y 381.301,Z 470.107,A -85,B 0,C 180,E1 -12126.079,E2 -12126.079} C_VEL
LIN {X 0,Y 381.336,Z 470.189,A -85,B 0,C 180,E1 -12127.231,E2 -12127.231} C_VEL
LIN {X 0,Y 381.299,Z 469.831,A -85,B 0,C 180,E1 -12128.37,E2 -12128.37} C_VEL
LIN {X 0,Y 381.426,Z 468.516,A -85,B 0,C 180,E1 -12129.986,E2 -12129.986} C_VEL
LIN {X 0,Y 381.639,Z 465.978,A -85,B 0,C 180,E1 -12131.757,E2 -12131.757} C_VEL
LIN {X 0,Y 381.876,Z 462.127,A -85,B 0,C 180,E1 -12133.567,E2 -12133.567} C_VEL
LIN {X 0,Y 382.212,Z 457.791,A -85,B 0,C 180,E1 -12135.084,E2 -12135.084} C_VEL
LIN {X 0,Y 382.73,Z 451.265,A -85,B 0,C 180,E1 -12136.86,E2 -12136.86} C_VEL
LIN {X 0,Y 383.327,Z 444.314,A -85,B 0,C 180,E1 -12138.366,E2 -12138.366} C_VEL
LIN {X 0,Y 384.236,Z 434.96,A -85,B 0,C 180,E1 -12139.994,E2 -12139.994} C_VEL
LIN {X 0,Y 385.139,Z 425.018,A -85,B 0,C 180,E1 -12141.367,E2 -12141.367} C_VEL
LIN {X 0,Y 386.069,Z 414.366,A -85,B 0,C 180,E1 -12142.548,E2 -12142.548} C_VEL
LIN {X 0,Y 386.943,Z 403.833,A -85,B 0,C 180,E1 -12143.483,E2 -12143.483} C_VEL
LIN {X 0,Y 387.669,Z 391.339,A -85,B 0,C 180,E1 -12144.344,E2 -12144.344} C_VEL
LIN {X 0,Y 388.284,Z 378.879,A -85,B 0,C 180,E1 -12144.97,E2 -12144.97} C_VEL
LIN {X 0,Y 388.814,Z 365.447,A -85,B 0,C 180,E1 -12145.416,E2 -12145.416} C_VEL
LIN {X 0,Y 389.919,Z 283.665,A -85,B 0,C 180,E1 -12146.97,E2 -12146.97} C_VEL
LIN {X 0,Y 388.534,Z 280.042,A -85,B 0,C 180,E1 -12147.112,E2 -12147.112} C_VEL
LIN {X 0,Y 381.067,Z 269.53,A -85,B 0,C 180,E1 -12147.707,E2 -12147.707} C_VEL
LIN {X 0,Y 379.781,Z 265.887,A -85,B 0,C 180,E1 -12147.849,E2 -12147.849} C_VEL
LIN {X 0,Y 378.557,Z 259.475,A -85,B 0,C 180,E1 -12148.073,E2 -12148.073} C_VEL
LIN {X 0,Y 378.76,Z 255.657,A -85,B 0,C 180,E1 -12148.938,E2 -12148.938} C_VEL
LIN {X 0,Y 378.408,Z 251.574,A -85,B 0,C 180,E1 -12150.001,E2 -12150.001} C_VEL
LIN {X 0,Y 376.327,Z 240.743,A -85,B 0,C 180,E1 -12152.945,E2 -12152.945} C_VEL
LIN {X 0,Y 376.158,Z 240.15,A -85,B 0,C 180,E1 -12153.214,E2 -12153.214} C_VEL
LIN {X 0,Y 376.205,Z 240.12,A -85,B 0,C 180,E1 -12156.437,E2 -12156.437} C_VEL
LIN {X 0,Y 376.086,Z 240.135,A -85,B 0,C 180,E1 -12159.683,E2 -12159.683} C_VEL
LIN {X 0,Y 376.056,Z 240.136,A -85,B 0,C 180,E1 -12163.66,E2 -12163.66} C_VEL
LIN {X 0,Y 376.01,Z 240.146,A -85,B 0,C 180,E1 -12167.609,E2 -12167.609} C_VEL
LIN {X 0,Y 375.947,Z 240.151,A -85,B 0,C 180,E1 -12170.835,E2 -12170.835} C_VEL
LIN {X 0,Y 375.944,Z 240.15,A -85,B 0,C 180,E1 -12174.286,E2 -12174.286} C_VEL
LIN {X 0,Y 375.905,Z 240.16,A -85,B 0,C 180,E1 -12177.867,E2 -12177.867} C_VEL
LIN {X 0,Y 375.91,Z 240.157,A -85,B 0,C 180,E1 -12181.567,E2 -12181.567} C_VEL
LIN {X 0,Y 375.947,Z 240.143,A -85,B 0,C 180,E1 -12184.669,E2 -12184.669} C_VEL
LIN {X 0,Y 375.909,Z 240.16,A -85,B 0,C 180,E1 -12188.266,E2 -12188.266} C_VEL
LIN {X 0,Y 375.889,Z 240.15,A -85,B 0,C 180,E1 -12191.601,E2 -12191.601} C_VEL
LIN {X 0,Y 375.899,Z 240.156,A -85,B 0,C 180,E1 -12194.734,E2 -12194.734} C_VEL
LIN {X 0,Y 375.887,Z 240.158,A -85,B 0,C 180,E1 -12197.7,E2 -12197.7} C_VEL
LIN {X 0,Y 375.915,Z 240.143,A -85,B 0,C 180,E1 -12200.538,E2 -12200.538} C_VEL
LIN {X 0,Y 375.941,Z 240.15,A -85,B 0,C 180,E1 -12203.501,E2 -12203.501} C_VEL
LIN {X 0,Y 375.942,Z 240.152,A -85,B 0,C 180,E1 -12205.892,E2 -12205.892} C_VEL
LIN {X 0,Y 375.947,Z 240.137,A -85,B 0,C 180,E1 -12209.691,E2 -12209.691} C_VEL
LIN {X 0,Y 375.905,Z 240.139,A -85,B 0,C 180,E1 -12212.139,E2 -12212.139} C_VEL
LIN {X 0,Y 375.948,Z 240.155,A -85,B 0,C 180,E1 -12215.72,E2 -12215.72} C_VEL
LIN {X 0,Y 375.991,Z 240.146,A -85,B 0,C 180,E1 -12219.202,E2 -12219.202} C_VEL
LIN {X 0,Y 376.026,Z 240.113,A -85,B 0,C 180,E1 -12222.604,E2 -12222.604} C_VEL
LIN {X 0,Y 376.086,Z 240.133,A -85,B 0,C 180,E1 -12226.347,E2 -12226.347} C_VEL
LIN {X 0,Y 376.106,Z 240.128,A -85,B 0,C 180,E1 -12230.322,E2 -12230.322} C_VEL
LIN {X 0,Y 376.192,Z 240.099,A -85,B 0,C 180,E1 -12233.568,E2 -12233.568} C_VEL
LIN {X 0,Y 376.339,Z 240.1,A -85,B 0,C 180,E1 -12237.863,E2 -12237.863} C_VEL
LIN {X 0,Y 376.335,Z 240.1,A -85,B 0,C 180,E1 -12242.144,E2 -12242.144} C_VEL
LIN {X 0,Y 376.221,Z 240.101,A -85,B 0,C 180,E1 -12246.439,E2 -12246.439} C_VEL
LIN {X 0,Y 376.117,Z 240.13,A -85,B 0,C 180,E1 -12249.685,E2 -12249.685} C_VEL
LIN {X 0,Y 376.097,Z 240.124,A -85,B 0,C 180,E1 -12253.66,E2 -12253.66} C_VEL
LIN {X 0,Y 376.041,Z 240.137,A -85,B 0,C 180,E1 -12257.403,E2 -12257.403} C_VEL
LIN {X 0,Y 375.988,Z 240.151,A -85,B 0,C 180,E1 -12260.835,E2 -12260.835} C_VEL
LIN {X 0,Y 375.982,Z 240.13,A -85,B 0,C 180,E1 -12264.285,E2 -12264.285} C_VEL
LIN {X 0,Y 375.939,Z 240.154,A -85,B 0,C 180,E1 -12267.866,E2 -12267.866} C_VEL
LIN {X 0,Y 375.967,Z 240.142,A -85,B 0,C 180,E1 -12271.564,E2 -12271.564} C_VEL
LIN {X 0,Y 375.967,Z 240.152,A -85,B 0,C 180,E1 -12275.418,E2 -12275.418} C_VEL
LIN {X 0,Y 375.947,Z 240.149,A -85,B 0,C 180,E1 -12278.264,E2 -12278.264} C_VEL
LIN {X 0,Y 375.929,Z 240.153,A -85,B 0,C 180,E1 -12281.599,E2 -12281.599} C_VEL
LIN {X 0,Y 375.935,Z 240.154,A -85,B 0,C 180,E1 -12284.732,E2 -12284.732} C_VEL
LIN {X 0,Y 375.938,Z 240.158,A -85,B 0,C 180,E1 -12287.7,E2 -12287.7} C_VEL
LIN {X 0,Y 375.946,Z 240.154,A -85,B 0,C 180,E1 -12290.535,E2 -12290.535} C_VEL
LIN {X 0,Y 375.975,Z 240.153,A -85,B 0,C 180,E1 -12293.497,E2 -12293.497} C_VEL
LIN {X 0,Y 375.973,Z 240.149,A -85,B 0,C 180,E1 -12295.889,E2 -12295.889} C_VEL
LIN {X 0,Y 375.977,Z 240.148,A -85,B 0,C 180,E1 -12299.688,E2 -12299.688} C_VEL
LIN {X 0,Y 376.022,Z 240.2,A -85,B 0,C 180,E1 -12301.811,E2 -12301.811} C_VEL
LIN {X 0,Y 377.02,Z 245.061,A -85,B 0,C 180,E1 -12303.155,E2 -12303.155} C_VEL
LIN {X 0,Y 379.141,Z 255.909,A -85,B 0,C 180,E1 -12305.932,E2 -12305.932} C_VEL
LIN {X 0,Y 379.016,Z 260.747,A -85,B 0,C 180,E1 -12307.082,E2 -12307.082} C_VEL
LIN {X 0,Y 378.343,Z 268.824,A -85,B 0,C 180,E1 -12308.932,E2 -12308.932} C_VEL
LIN {X 0,Y 381.12,Z 284.999,A -85,B 0,C 180,E1 -12309.444,E2 -12309.444} C_VEL
LIN {X 0,Y 383.266,Z 299.083,A -85,B 0,C 180,E1 -12309.837,E2 -12309.837} C_VEL
LIN {X 0,Y 381.962,Z 377.384,A -85,B 0,C 180,E1 -12311.355,E2 -12311.355} C_VEL
LIN {X 0,Y 381.319,Z 391.1,A -85,B 0,C 180,E1 -12311.844,E2 -12311.844} C_VEL
LIN {X 0,Y 380.577,Z 403.965,A -85,B 0,C 180,E1 -12312.537,E2 -12312.537} C_VEL
LIN {X 0,Y 379.6,Z 416.506,A -85,B 0,C 180,E1 -12313.461,E2 -12313.461} C_VEL
LIN {X 0,Y 378.646,Z 427.699,A -85,B 0,C 180,E1 -12314.525,E2 -12314.525} C_VEL
LIN {X 0,Y 377.706,Z 438.363,A -85,B 0,C 180,E1 -12315.811,E2 -12315.811} C_VEL
LIN {X 0,Y 376.734,Z 448.501,A -85,B 0,C 180,E1 -12317.337,E2 -12317.337} C_VEL
LIN {X 0,Y 375.91,Z 457.029,A -85,B 0,C 180,E1 -12318.951,E2 -12318.951} C_VEL
LIN {X 0,Y 375.325,Z 463.867,A -85,B 0,C 180,E1 -12320.569,E2 -12320.569} C_VEL
LIN {X 0,Y 374.852,Z 470.144,A -85,B 0,C 180,E1 -12322.458,E2 -12322.458} C_VEL
LIN {X 0,Y 374.608,Z 473.844,A -85,B 0,C 180,E1 -12323.911,E2 -12323.911} C_VEL
LIN {X 0,Y 374.532,Z 477.249,A -85,B 0,C 180,E1 -12325.695,E2 -12325.695} C_VEL
LIN {X 0,Y 374.437,Z 478.73,A -85,B 0,C 180,E1 -12326.771,E2 -12326.771} C_VEL
LIN {X 0,Y 374.457,Z 480.419,A -85,B 0,C 180,E1 -12328.924,E2 -12328.924} C_VEL
LIN {X 0,Y 374.478,Z 480.681,A -85,B 0,C 180,E1 -12329.999,E2 -12329.999} C_VEL
LIN {X 0,Y 374.456,Z 480.536,A -85,B 0,C 180,E1 -12331.075,E2 -12331.075} C_VEL
LIN {X 0,Y 374.438,Z 479.004,A -85,B 0,C 180,E1 -12333.227,E2 -12333.227} C_VEL
LIN {X 0,Y 374.562,Z 477.65,A -85,B 0,C 180,E1 -12334.303,E2 -12334.303} C_VEL
LIN {X 0,Y 374.648,Z 474.326,A -85,B 0,C 180,E1 -12336.146,E2 -12336.146} C_VEL
LIN {X 0,Y 374.987,Z 469.341,A -85,B 0,C 180,E1 -12338.08,E2 -12338.08} C_VEL
LIN {X 0,Y 375.544,Z 462.894,A -85,B 0,C 180,E1 -12339.967,E2 -12339.967} C_VEL
LIN {X 0,Y 376.198,Z 455.85,A -85,B 0,C 180,E1 -12341.584,E2 -12341.584} C_VEL
LIN {X 0,Y 377.195,Z 447.047,A -85,B 0,C 180,E1 -12343.193,E2 -12343.193} C_VEL
LIN {X 0,Y 378.116,Z 437.557,A -85,B 0,C 180,E1 -12344.599,E2 -12344.599} C_VEL
LIN {X 0,Y 379.126,Z 426.871,A -85,B 0,C 180,E1 -12345.867,E2 -12345.867} C_VEL
LIN {X 0,Y 380.214,Z 415.58,A -85,B 0,C 180,E1 -12346.924,E2 -12346.924} C_VEL
LIN {X 0,Y 381.159,Z 403.884,A -85,B 0,C 180,E1 -12347.78,E2 -12347.78} C_VEL
LIN {X 0,Y 382.024,Z 391.14,A -85,B 0,C 180,E1 -12348.467,E2 -12348.467} C_VEL
LIN {X 0,Y 382.663,Z 377.62,A -85,B 0,C 180,E1 -12348.955,E2 -12348.955} C_VEL
LIN {X 0,Y 383.489,Z 333.301,A -85,B 0,C 180,E1 -12349.836,E2 -12349.836} C_VEL
LIN {X 0,Y 383.911,Z 297.869,A -85,B 0,C 180,E1 -12350.527,E2 -12350.527} C_VEL
LIN {X 0,Y 380.002,Z 275.372,A -85,B 0,C 180,E1 -12351.224,E2 -12351.224} C_VEL
LIN {X 0,Y 378.689,Z 268.533,A -85,B 0,C 180,E1 -12351.492,E2 -12351.492} C_VEL
LIN {X 0,Y 379.527,Z 258.455,A -85,B 0,C 180,E1 -12353.75,E2 -12353.75} C_VEL
LIN {X 0,Y 377.884,Z 248.692,A -85,B 0,C 180,E1 -12356.212,E2 -12356.212} C_VEL
LIN {X 0,Y 376.04,Z 240.407,A -85,B 0,C 180,E1 -12358.423,E2 -12358.423} C_VEL
LIN {X 0,Y 375.968,Z 240.156,A -85,B 0,C 180,E1 -12359.078,E2 -12359.078} C_VEL
LIN {X 0,Y 375.956,Z 240.155,A -85,B 0,C 180,E1 -12362.826,E2 -12362.826} C_VEL
LIN {X 0,Y 375.962,Z 240.155,A -85,B 0,C 180,E1 -12365.414,E2 -12365.414} C_VEL
LIN {X 0,Y 375.941,Z 240.158,A -85,B 0,C 180,E1 -12368.261,E2 -12368.261} C_VEL
LIN {X 0,Y 375.923,Z 240.155,A -85,B 0,C 180,E1 -12371.596,E2 -12371.596} C_VEL
LIN {X 0,Y 375.93,Z 240.157,A -85,B 0,C 180,E1 -12374.729,E2 -12374.729} C_VEL
LIN {X 0,Y 375.929,Z 240.157,A -85,B 0,C 180,E1 -12377.696,E2 -12377.696} C_VEL
LIN {X 0,Y 375.937,Z 240.156,A -85,B 0,C 180,E1 -12380.531,E2 -12380.531} C_VEL
LIN {X 0,Y 375.96,Z 240.151,A -85,B 0,C 180,E1 -12383.494,E2 -12383.494} C_VEL
LIN {X 0,Y 375.959,Z 240.15,A -85,B 0,C 180,E1 -12385.885,E2 -12385.885} C_VEL
LIN {X 0,Y 375.962,Z 240.149,A -85,B 0,C 180,E1 -12389.684,E2 -12389.684} C_VEL
LIN {X 0,Y 375.918,Z 240.155,A -85,B 0,C 180,E1 -12392.132,E2 -12392.132} C_VEL
LIN {X 0,Y 375.967,Z 240.149,A -85,B 0,C 180,E1 -12395.714,E2 -12395.714} C_VEL
LIN {X 0,Y 375.997,Z 240.15,A -85,B 0,C 180,E1 -12399.195,E2 -12399.195} C_VEL
LIN {X 0,Y 376.03,Z 240.137,A -85,B 0,C 180,E1 -12402.597,E2 -12402.597} C_VEL
LIN {X 0,Y 376.086,Z 240.129,A -85,B 0,C 180,E1 -12406.339,E2 -12406.339} C_VEL
LIN {X 0,Y 376.104,Z 240.131,A -85,B 0,C 180,E1 -12410.315,E2 -12410.315} C_VEL
LIN {X 0,Y 376.211,Z 240.125,A -85,B 0,C 180,E1 -12413.561,E2 -12413.561} C_VEL
LIN {X 0,Y 376.322,Z 240.109,A -85,B 0,C 180,E1 -12417.856,E2 -12417.856} C_VEL
LIN {X 0,Y 376.32,Z 240.107,A -85,B 0,C 180,E1 -12422.137,E2 -12422.137} C_VEL
LIN {X 0,Y 376.177,Z 240.123,A -85,B 0,C 180,E1 -12426.432,E2 -12426.432} C_VEL
LIN {X 0,Y 376.093,Z 240.133,A -85,B 0,C 180,E1 -12429.678,E2 -12429.678} C_VEL
LIN {X 0,Y 376.075,Z 240.136,A -85,B 0,C 180,E1 -12433.654,E2 -12433.654} C_VEL
LIN {X 0,Y 376.016,Z 240.141,A -85,B 0,C 180,E1 -12437.396,E2 -12437.396} C_VEL
LIN {X 0,Y 375.96,Z 240.152,A -85,B 0,C 180,E1 -12440.828,E2 -12440.828} C_VEL
LIN {X 0,Y 375.958,Z 240.157,A -85,B 0,C 180,E1 -12444.279,E2 -12444.279} C_VEL
LIN {X 0,Y 375.913,Z 240.156,A -85,B 0,C 180,E1 -12447.86,E2 -12447.86} C_VEL
LIN {X 0,Y 375.934,Z 240.154,A -85,B 0,C 180,E1 -12451.559,E2 -12451.559} C_VEL
LIN {X 0,Y 375.933,Z 240.154,A -85,B 0,C 180,E1 -12455.412,E2 -12455.412} C_VEL
LIN {X 0,Y 375.952,Z 240.156,A -85,B 0,C 180,E1 -12458.268,E2 -12458.268} C_VEL
LIN {X 0,Y 375.993,Z 240.194,A -85,B 0,C 180,E1 -12460.73,E2 -12460.73} C_VEL
LIN {X 0,Y 377.59,Z 247.658,A -85,B 0,C 180,E1 -12462.787,E2 -12462.787} C_VEL
LIN {X 0,Y 379.072,Z 255.472,A -85,B 0,C 180,E1 -12464.784,E2 -12464.784} C_VEL
LIN {X 0,Y 378.958,Z 259.039,A -85,B 0,C 180,E1 -12465.578,E2 -12465.578} C_VEL
LIN {X 0,Y 382.864,Z 278.262,A -85,B 0,C 180,E1 -12466.254,E2 -12466.254} C_VEL
LIN {X 0,Y 384.169,Z 286.245,A -85,B 0,C 180,E1 -12466.495,E2 -12466.495} C_VEL
LIN {X 0,Y 382.697,Z 366.986,A -85,B 0,C 180,E1 -12468.066,E2 -12468.066} C_VEL
LIN {X 0,Y 382.124,Z 380.357,A -85,B 0,C 180,E1 -12468.541,E2 -12468.541} C_VEL
LIN {X 0,Y 381.462,Z 392.839,A -85,B 0,C 180,E1 -12469.202,E2 -12469.202} C_VEL
LIN {X 0,Y 380.577,Z 405.02,A -85,B 0,C 180,E1 -12470.082,E2 -12470.082} C_VEL
LIN {X 0,Y 379.528,Z 416.279,A -85,B 0,C 180,E1 -12471.128,E2 -12471.128} C_VEL
LIN {X 0,Y 378.605,Z 425.756,A -85,B 0,C 180,E1 -12472.226,E2 -12472.226} C_VEL
LIN {X 0,Y 377.698,Z 434.496,A -85,B 0,C 180,E1 -12473.458,E2 -12473.458} C_VEL
LIN {X 0,Y 376.795,Z 443.263,A -85,B 0,C 180,E1 -12474.978,E2 -12474.978} C_VEL
LIN {X 0,Y 376.046,Z 450.534,A -85,B 0,C 180,E1 -12476.543,E2 -12476.543} C_VEL
LIN {X 0,Y 375.363,Z 457.33,A -85,B 0,C 180,E1 -12478.384,E2 -12478.384} C_VEL
LIN {X 0,Y 374.921,Z 462.487,A -85,B 0,C 180,E1 -12480.216,E2 -12480.216} C_VEL
LIN {X 0,Y 374.597,Z 466.211,A -85,B 0,C 180,E1 -12482.029,E2 -12482.029} C_VEL
LIN {X 0,Y 374.409,Z 467.996,A -85,B 0,C 180,E1 -12483.225,E2 -12483.225} C_VEL
LIN {X 0,Y 374.314,Z 469.271,A -85,B 0,C 180,E1 -12484.417,E2 -12484.417} C_VEL
LIN {X 0,Y 374.214,Z 470.016,A -85,B 0,C 180,E1 -12485.597,E2 -12485.597} C_VEL
LIN {X 0,Y 374.244,Z 470.328,A -85,B 0,C 180,E1 -12486.938,E2 -12486.938} C_VEL
LIN {X 0,Y 374.22,Z 470.127,A -85,B 0,C 180,E1 -12487.939,E2 -12487.939} C_VEL
LIN {X 0,Y 374.309,Z 468.813,A -85,B 0,C 180,E1 -12489.834,E2 -12489.834} C_VEL
LIN {X 0,Y 374.573,Z 465.844,A -85,B 0,C 180,E1 -12491.967,E2 -12491.967} C_VEL
LIN {X 0,Y 374.795,Z 462.242,A -85,B 0,C 180,E1 -12493.665,E2 -12493.665} C_VEL
LIN {X 0,Y 375.181,Z 457.456,A -85,B 0,C 180,E1 -12495.353,E2 -12495.353} C_VEL
LIN {X 0,Y 375.714,Z 451.347,A -85,B 0,C 180,E1 -12497.029,E2 -12497.029} C_VEL
LIN {X 0,Y 376.407,Z 443.724,A -85,B 0,C 180,E1 -12498.695,E2 -12498.695} C_VEL
LIN {X 0,Y 377.213,Z 435.911,A -85,B 0,C 180,E1 -12500.077,E2 -12500.077} C_VEL
LIN {X 0,Y 378.11,Z 426.428,A -85,B 0,C 180,E1 -12501.45,E2 -12501.45} C_VEL
LIN {X 0,Y 379.076,Z 415.808,A -85,B 0,C 180,E1 -12502.678,E2 -12502.678} C_VEL
LIN {X 0,Y 380.088,Z 403.961,A -85,B 0,C 180,E1 -12503.765,E2 -12503.765} C_VEL
LIN {X 0,Y 380.873,Z 391.447,A -85,B 0,C 180,E1 -12504.641,E2 -12504.641} C_VEL
LIN {X 0,Y 381.492,Z 379.052,A -85,B 0,C 180,E1 -12505.276,E2 -12505.276} C_VEL
LIN {X 0,Y 382.036,Z 365.816,A -85,B 0,C 180,E1 -12505.726,E2 -12505.726} C_VEL
LIN {X 0,Y 383.207,Z 284.393,A -85,B 0,C 180,E1 -12507.298,E2 -12507.298} C_VEL
LIN {X 0,Y 379.781,Z 265.887,A -85,B 0,C 180,E1 -12507.849,E2 -12507.849} C_VEL
LIN {X 0,Y 378.877,Z 262.509,A -85,B 0,C 180,E1 -12508.046,E2 -12508.046} C_VEL
LIN {X 0,Y 377.278,Z 259.046,A -85,B 0,C 180,E1 -12508.473,E2 -12508.473} C_VEL
LIN {X 0,Y 374.804,Z 255.351,A -85,B 0,C 180,E1 -12509.259,E2 -12509.259} C_VEL
LIN {X 0,Y 372.113,Z 251.732,A -85,B 0,C 180,E1 -12510.369,E2 -12510.369} C_VEL
LIN {X 0,Y 370.534,Z 247.731,A -85,B 0,C 180,E1 -12511.523,E2 -12511.523} C_VEL
LIN {X 0,Y 369.113,Z 241.141,A -85,B 0,C 180,E1 -12513.412,E2 -12513.412} C_VEL
LIN {X 0,Y 369.165,Z 240.996,A -85,B 0,C 180,E1 -12516.56,E2 -12516.56} C_VEL
LIN {X 0,Y 369.035,Z 241.014,A -85,B 0,C 180,E1 -12519.87,E2 -12519.87} C_VEL
LIN {X 0,Y 369.004,Z 241.016,A -85,B 0,C 180,E1 -12523.774,E2 -12523.774} C_VEL
LIN {X 0,Y 368.969,Z 241.025,A -85,B 0,C 180,E1 -12527.771,E2 -12527.771} C_VEL
LIN {X 0,Y 368.878,Z 241.032,A -85,B 0,C 180,E1 -12531.224,E2 -12531.224} C_VEL
LIN {X 0,Y 368.899,Z 241.028,A -85,B 0,C 180,E1 -12534.78,E2 -12534.78} C_VEL
LIN {X 0,Y 368.887,Z 241.026,A -85,B 0,C 180,E1 -12538.445,E2 -12538.445} C_VEL
LIN {X 0,Y 368.863,Z 241.04,A -85,B 0,C 180,E1 -12542.242,E2 -12542.242} C_VEL
LIN {X 0,Y 368.896,Z 241.019,A -85,B 0,C 180,E1 -12545.003,E2 -12545.003} C_VEL
LIN {X 0,Y 368.851,Z 241.042,A -85,B 0,C 180,E1 -12548.637,E2 -12548.637} C_VEL
LIN {X 0,Y 368.835,Z 241.029,A -85,B 0,C 180,E1 -12552.009,E2 -12552.009} C_VEL
LIN {X 0,Y 368.852,Z 241.037,A -85,B 0,C 180,E1 -12555.179,E2 -12555.179} C_VEL
LIN {X 0,Y 368.84,Z 241.037,A -85,B 0,C 180,E1 -12558.178,E2 -12558.178} C_VEL
LIN {X 0,Y 368.858,Z 241.017,A -85,B 0,C 180,E1 -12561.37,E2 -12561.37} C_VEL
LIN {X 0,Y 368.915,Z 241.032,A -85,B 0,C 180,E1 -12565.15,E2 -12565.15} C_VEL
LIN {X 0,Y 368.882,Z 241.024,A -85,B 0,C 180,E1 -12569.048,E2 -12569.048} C_VEL
LIN {X 0,Y 368.894,Z 241.009,A -85,B 0,C 180,E1 -12571.562,E2 -12571.562} C_VEL
LIN {X 0,Y 368.887,Z 241.031,A -85,B 0,C 180,E1 -12575.225,E2 -12575.225} C_VEL
LIN {X 0,Y 368.91,Z 241.031,A -85,B 0,C 180,E1 -12577.608,E2 -12577.608} C_VEL
LIN {X 0,Y 368.947,Z 241.008,A -85,B 0,C 180,E1 -12581.11,E2 -12581.11} C_VEL
LIN {X 0,Y 368.992,Z 241.006,A -85,B 0,C 180,E1 -12584.539,E2 -12584.539} C_VEL
LIN {X 0,Y 369.053,Z 241.008,A -85,B 0,C 180,E1 -12586.794,E2 -12586.794} C_VEL
LIN {X 0,Y 369.056,Z 241.007,A -85,B 0,C 180,E1 -12590.136,E2 -12590.136} C_VEL
LIN {X 0,Y 369.154,Z 240.976,A -85,B 0,C 180,E1 -12593.445,E2 -12593.445} C_VEL
LIN {X 0,Y 369.303,Z 240.976,A -85,B 0,C 180,E1 -12597.823,E2 -12597.823} C_VEL
LIN {X 0,Y 369.298,Z 240.976,A -85,B 0,C 180,E1 -12602.185,E2 -12602.185} C_VEL
LIN {X 0,Y 369.182,Z 240.979,A -85,B 0,C 180,E1 -12606.562,E2 -12606.562} C_VEL
LIN {X 0,Y 369.067,Z 241.009,A -85,B 0,C 180,E1 -12609.872,E2 -12609.872} C_VEL
LIN {X 0,Y 369.045,Z 241.002,A -85,B 0,C 180,E1 -12613.775,E2 -12613.775} C_VEL
LIN {X 0,Y 369,Z 241.013,A -85,B 0,C 180,E1 -12617.746,E2 -12617.746} C_VEL
LIN {X 0,Y 368.919,Z 241.027,A -85,B 0,C 180,E1 -12621.223,E2 -12621.223} C_VEL
LIN {X 0,Y 368.936,Z 241.011,A -85,B 0,C 180,E1 -12624.78,E2 -12624.78} C_VEL
LIN {X 0,Y 368.923,Z 241.028,A -85,B 0,C 180,E1 -12628.444,E2 -12628.444} C_VEL
LIN {X 0,Y 368.908,Z 241.022,A -85,B 0,C 180,E1 -12632.24,E2 -12632.24} C_VEL
LIN {X 0,Y 368.939,Z 241.029,A -85,B 0,C 180,E1 -12635.003,E2 -12635.003} C_VEL
LIN {X 0,Y 368.888,Z 241.028,A -85,B 0,C 180,E1 -12638.635,E2 -12638.635} C_VEL
LIN {X 0,Y 368.882,Z 241.026,A -85,B 0,C 180,E1 -12642.009,E2 -12642.009} C_VEL
LIN {X 0,Y 368.887,Z 241.035,A -85,B 0,C 180,E1 -12645.176,E2 -12645.176} C_VEL
LIN {X 0,Y 368.881,Z 241.035,A -85,B 0,C 180,E1 -12648.177,E2 -12648.177} C_VEL
LIN {X 0,Y 368.889,Z 241.035,A -85,B 0,C 180,E1 -12651.367,E2 -12651.367} C_VEL
LIN {X 0,Y 368.949,Z 241.027,A -85,B 0,C 180,E1 -12655.147,E2 -12655.147} C_VEL
LIN {X 0,Y 368.943,Z 241.024,A -85,B 0,C 180,E1 -12659.047,E2 -12659.047} C_VEL
LIN {X 0,Y 368.973,Z 241.175,A -85,B 0,C 180,E1 -12661.563,E2 -12661.563} C_VEL
LIN {X 0,Y 371.191,Z 251.954,A -85,B 0,C 180,E1 -12664.465,E2 -12664.465} C_VEL
LIN {X 0,Y 372.303,Z 258.125,A -85,B 0,C 180,E1 -12666.054,E2 -12666.054} C_VEL
LIN {X 0,Y 371.469,Z 268.689,A -85,B 0,C 180,E1 -12668.54,E2 -12668.54} C_VEL
LIN {X 0,Y 372.541,Z 275.002,A -85,B 0,C 180,E1 -12668.777,E2 -12668.777} C_VEL
LIN {X 0,Y 376.547,Z 299.16,A -85,B 0,C 180,E1 -12669.488,E2 -12669.488} C_VEL
LIN {X 0,Y 375.236,Z 376.441,A -85,B 0,C 180,E1 -12671.008,E2 -12671.008} C_VEL
LIN {X 0,Y 374.634,Z 389.678,A -85,B 0,C 180,E1 -12671.473,E2 -12671.473} C_VEL
LIN {X 0,Y 373.839,Z 402.41,A -85,B 0,C 180,E1 -12672.141,E2 -12672.141} C_VEL
LIN {X 0,Y 372.899,Z 414.533,A -85,B 0,C 180,E1 -12673.014,E2 -12673.014} C_VEL
LIN {X 0,Y 371.879,Z 426.074,A -85,B 0,C 180,E1 -12674.095,E2 -12674.095} C_VEL
LIN {X 0,Y 371.029,Z 435.552,A -85,B 0,C 180,E1 -12675.203,E2 -12675.203} C_VEL
LIN {X 0,Y 370.169,Z 444.976,A -85,B 0,C 180,E1 -12676.55,E2 -12676.55} C_VEL
LIN {X 0,Y 369.146,Z 454.171,A -85,B 0,C 180,E1 -12678.189,E2 -12678.189} C_VEL
LIN {X 0,Y 368.488,Z 461.572,A -85,B 0,C 180,E1 -12679.838,E2 -12679.838} C_VEL
LIN {X 0,Y 367.912,Z 468.362,A -85,B 0,C 180,E1 -12681.762,E2 -12681.762} C_VEL
LIN {X 0,Y 367.593,Z 472.835,A -85,B 0,C 180,E1 -12683.412,E2 -12683.412} C_VEL
LIN {X 0,Y 367.49,Z 475.194,A -85,B 0,C 180,E1 -12684.512,E2 -12684.512} C_VEL
LIN {X 0,Y 367.442,Z 477.12,A -85,B 0,C 180,E1 -12685.611,E2 -12685.611} C_VEL
LIN {X 0,Y 367.357,Z 478.613,A -85,B 0,C 180,E1 -12686.709,E2 -12686.709} C_VEL
LIN {X 0,Y 367.355,Z 480.312,A -85,B 0,C 180,E1 -12688.903,E2 -12688.903} C_VEL
LIN {X 0,Y 367.379,Z 480.579,A -85,B 0,C 180,E1 -12689.999,E2 -12689.999} C_VEL
LIN {X 0,Y 367.355,Z 480.444,A -85,B 0,C 180,E1 -12691.095,E2 -12691.095} C_VEL
LIN {X 0,Y 367.359,Z 478.924,A -85,B 0,C 180,E1 -12693.289,E2 -12693.289} C_VEL
LIN {X 0,Y 367.471,Z 477.576,A -85,B 0,C 180,E1 -12694.387,E2 -12694.387} C_VEL
LIN {X 0,Y 367.551,Z 474.589,A -85,B 0,C 180,E1 -12696.105,E2 -12696.105} C_VEL
LIN {X 0,Y 367.828,Z 470.846,A -85,B 0,C 180,E1 -12697.685,E2 -12697.685} C_VEL
LIN {X 0,Y 368.257,Z 465.842,A -85,B 0,C 180,E1 -12699.335,E2 -12699.335} C_VEL
LIN {X 0,Y 368.901,Z 459.561,A -85,B 0,C 180,E1 -12700.982,E2 -12700.982} C_VEL
LIN {X 0,Y 369.73,Z 451.702,A -85,B 0,C 180,E1 -12702.626,E2 -12702.626} C_VEL
LIN {X 0,Y 370.852,Z 441.91,A -85,B 0,C 180,E1 -12704.261,E2 -12704.261} C_VEL
LIN {X 0,Y 371.812,Z 431.74,A -85,B 0,C 180,E1 -12705.625,E2 -12705.625} C_VEL
LIN {X 0,Y 372.896,Z 421.668,A -85,B 0,C 180,E1 -12706.702,E2 -12706.702} C_VEL
LIN {X 0,Y 373.889,Z 410.712,A -85,B 0,C 180,E1 -12707.643,E2 -12707.643} C_VEL
LIN {X 0,Y 374.835,Z 398.605,A -85,B 0,C 180,E1 -12708.444,E2 -12708.444} C_VEL
LIN {X 0,Y 375.617,Z 386.074,A -85,B 0,C 180,E1 -12709.041,E2 -12709.041} C_VEL
LIN {X 0,Y 376.13,Z 373.067,A -85,B 0,C 180,E1 -12709.439,E2 -12709.439} C_VEL
LIN {X 0,Y 377.354,Z 299.021,A -85,B 0,C 180,E1 -12710.898,E2 -12710.898} C_VEL
LIN {X 0,Y 373.516,Z 276.797,A -85,B 0,C 180,E1 -12711.606,E2 -12711.606} C_VEL
LIN {X 0,Y 371.889,Z 268.624,A -85,B 0,C 180,E1 -12711.916,E2 -12711.916} C_VEL
LIN {X 0,Y 372.05,Z 265.793,A -85,B 0,C 180,E1 -12712.489,E2 -12712.489} C_VEL
LIN {X 0,Y 372.617,Z 259.69,A -85,B 0,C 180,E1 -12713.922,E2 -12713.922} C_VEL
LIN {X 0,Y 370.964,Z 250.048,A -85,B 0,C 180,E1 -12716.41,E2 -12716.41} C_VEL
LIN {X 0,Y 368.952,Z 241.151,A -85,B 0,C 180,E1 -12718.874,E2 -12718.874} C_VEL
LIN {X 0,Y 368.904,Z 241.033,A -85,B 0,C 180,E1 -12722.236,E2 -12722.236} C_VEL
LIN {X 0,Y 368.935,Z 241.029,A -85,B 0,C 180,E1 -12724.999,E2 -12724.999} C_VEL
LIN {X 0,Y 368.882,Z 241.034,A -85,B 0,C 180,E1 -12728.632,E2 -12728.632} C_VEL
LIN {X 0,Y 368.876,Z 241.037,A -85,B 0,C 180,E1 -12732.005,E2 -12732.005} C_VEL
LIN {X 0,Y 368.882,Z 241.032,A -85,B 0,C 180,E1 -12735.173,E2 -12735.173} C_VEL
LIN {X 0,Y 368.874,Z 241.035,A -85,B 0,C 180,E1 -12738.173,E2 -12738.173} C_VEL
LIN {X 0,Y 368.879,Z 241.029,A -85,B 0,C 180,E1 -12741.363,E2 -12741.363} C_VEL
LIN {X 0,Y 368.932,Z 241.025,A -85,B 0,C 180,E1 -12745.143,E2 -12745.143} C_VEL
LIN {X 0,Y 368.914,Z 241.028,A -85,B 0,C 180,E1 -12749.042,E2 -12749.042} C_VEL
LIN {X 0,Y 368.908,Z 241.028,A -85,B 0,C 180,E1 -12751.555,E2 -12751.555} C_VEL
LIN {X 0,Y 368.922,Z 241.029,A -85,B 0,C 180,E1 -12755.219,E2 -12755.219} C_VEL
LIN {X 0,Y 368.919,Z 241.032,A -85,B 0,C 180,E1 -12758.977,E2 -12758.977} C_VEL
LIN {X 0,Y 368.989,Z 241.012,A -85,B 0,C 180,E1 -12762.254,E2 -12762.254} C_VEL
LIN {X 0,Y 369.034,Z 241.007,A -85,B 0,C 180,E1 -12766.224,E2 -12766.224} C_VEL
LIN {X 0,Y 369.054,Z 241.009,A -85,B 0,C 180,E1 -12770.128,E2 -12770.128} C_VEL
LIN {X 0,Y 369.171,Z 241.001,A -85,B 0,C 180,E1 -12773.438,E2 -12773.438} C_VEL
LIN {X 0,Y 369.286,Z 240.986,A -85,B 0,C 180,E1 -12777.815,E2 -12777.815} C_VEL
LIN {X 0,Y 369.283,Z 240.983,A -85,B 0,C 180,E1 -12782.178,E2 -12782.178} C_VEL
LIN {X 0,Y 369.139,Z 241,A -85,B 0,C 180,E1 -12786.555,E2 -12786.555} C_VEL
